LIN {X 0,Y 530.48,Z 461.696,A -85,B 0,C 180,E1 -4342.594,E2 -4342.594} C_VEL
LIN {X 0,Y 530.522,Z 458.64,A -85,B 0,C 180,E1 -4345.082,E2 -4345.082} C_VEL
LIN {X 0,Y 530.512,Z 455.242,A -85,B 0,C 180,E1 -4347.624,E2 -4347.624} C_VEL
LIN {X 0,Y 530.476,Z 451.107,A -85,B 0,C 180,E1 -4350.553,E2 -4350.553} C_VEL
LIN {X 0,Y 530.495,Z 450.409,A -85,B 0,C 180,E1 -4351.109,E2 -4351.109} C_VEL
LIN {X 0,Y 530.816,Z 450.368,A -85,B 0,C 180,E1 -4353.785,E2 -4353.785} C_VEL
LIN {X 0,Y 530.957,Z 450.348,A -85,B 0,C 180,E1 -4356.558,E2 -4356.558} C_VEL
LIN {X 0,Y 530.988,Z 450.346,A -85,B 0,C 180,E1 -4359.443,E2 -4359.443} C_VEL
LIN {X 0,Y 530.985,Z 450.345,A -85,B 0,C 180,E1 -4362.456,E2 -4362.456} C_VEL
LIN {X 0,Y 530.991,Z 450.345,A -85,B 0,C 180,E1 -4365.621,E2 -4365.621} C_VEL
LIN {X 0,Y 530.999,Z 450.345,A -85,B 0,C 180,E1 -4368.565,E2 -4368.565} C_VEL
LIN {X 0,Y 530.986,Z 450.347,A -85,B 0,C 180,E1 -4371.653,E2 -4371.653} C_VEL
LIN {X 0,Y 531.348,Z 452.371,A -85,B 0,C 180,E1 -4372.524,E2 -4372.524} C_VEL
LIN {X 0,Y 532.063,Z 457.513,A -85,B 0,C 180,E1 -4374.465,E2 -4374.465} C_VEL
LIN {X 0,Y 531.885,Z 464.036,A -85,B 0,C 180,E1 -4376.765,E2 -4376.765} C_VEL
LIN {X 0,Y 531.715,Z 471.225,A -85,B 0,C 180,E1 -4379.221,E2 -4379.221} C_VEL
LIN {X 0,Y 531.434,Z 481.002,A -85,B 0,C 180,E1 -4382.428,E2 -4382.428} C_VEL
LIN {X 0,Y 531.236,Z 490.287,A -85,B 0,C 180,E1 -4385.372,E2 -4385.372} C_VEL
LIN {X 0,Y 531.041,Z 500.911,A -85,B 0,C 180,E1 -4388.657,E2 -4388.657} C_VEL
LIN {X 0,Y 530.899,Z 510.447,A -85,B 0,C 180,E1 -4391.475,E2 -4391.475} C_VEL
LIN {X 0,Y 530.798,Z 519.953,A -85,B 0,C 180,E1 -4394.251,E2 -4394.251} C_VEL
LIN {X 0,Y 530.709,Z 527.53,A -85,B 0,C 180,E1 -4396.454,E2 -4396.454} C_VEL
LIN {X 0,Y 532.33,Z 538.348,A -85,B 0,C 180,E1 -4396.739,E2 -4396.739} C_VEL
LIN {X 0,Y 532.122,Z 551.772,A -85,B 0,C 180,E1 -4397.17,E2 -4397.17} C_VEL
LIN {X 0,Y 531.932,Z 563.405,A -85,B 0,C 180,E1 -4397.699,E2 -4397.699} C_VEL
LIN {X 0,Y 531.637,Z 575.806,A -85,B 0,C 180,E1 -4398.441,E2 -4398.441} C_VEL
LIN {X 0,Y 531.384,Z 586.265,A -85,B 0,C 180,E1 -4399.233,E2 -4399.233} C_VEL
LIN {X 0,Y 531.113,Z 595.539,A -85,B 0,C 180,E1 -4400.094,E2 -4400.094} C_VEL
LIN {X 0,Y 530.931,Z 603.991,A -85,B 0,C 180,E1 -4401.052,E2 -4401.052} C_VEL
LIN {X 0,Y 530.758,Z 612.235,A -85,B 0,C 180,E1 -4402.199,E2 -4402.199} C_VEL
LIN {X 0,Y 530.598,Z 619.269,A -85,B 0,C 180,E1 -4403.419,E2 -4403.419} C_VEL
LIN {X 0,Y 530.525,Z 624.949,A -85,B 0,C 180,E1 -4404.679,E2 -4404.679} C_VEL
LIN {X 0,Y 530.522,Z 628.894,A -85,B 0,C 180,E1 -4405.822,E2 -4405.822} C_VEL
LIN {X 0,Y 530.457,Z 631.807,A -85,B 0,C 180,E1 -4406.962,E2 -4406.962} C_VEL
LIN {X 0,Y 530.41,Z 633.194,A -85,B 0,C 180,E1 -4407.722,E2 -4407.722} C_VEL
LIN {X 0,Y 530.344,Z 634.786,A -85,B 0,C 180,E1 -4409.241,E2 -4409.241} C_VEL
LIN {X 0,Y 530.342,Z 635,A -85,B 0,C 180,E1 -4410,E2 -4410} C_VEL
LIN {X 0,Y 530.361,Z 634.184,A -85,B 0,C 180,E1 -4411.519,E2 -4411.519} C_VEL
LIN {X 0,Y 530.41,Z 633.196,A -85,B 0,C 180,E1 -4412.278,E2 -4412.278} C_VEL
LIN {X 0,Y 530.457,Z 631.81,A -85,B 0,C 180,E1 -4413.038,E2 -4413.038} C_VEL
LIN {X 0,Y 530.522,Z 628.895,A -85,B 0,C 180,E1 -4414.178,E2 -4414.178} C_VEL
LIN {X 0,Y 530.525,Z 624.948,A -85,B 0,C 180,E1 -4415.321,E2 -4415.321} C_VEL
LIN {X 0,Y 530.599,Z 619.262,A -85,B 0,C 180,E1 -4416.582,E2 -4416.582} C_VEL
LIN {X 0,Y 530.758,Z 612.235,A -85,B 0,C 180,E1 -4417.801,E2 -4417.801} C_VEL
LIN {X 0,Y 530.931,Z 603.992,A -85,B 0,C 180,E1 -4418.948,E2 -4418.948} C_VEL
LIN {X 0,Y 531.113,Z 595.539,A -85,B 0,C 180,E1 -4419.906,E2 -4419.906} C_VEL
LIN {X 0,Y 531.407,Z 585.091,A -85,B 0,C 180,E1 -4420.863,E2 -4420.863} C_VEL
LIN {X 0,Y 531.675,Z 574.17,A -85,B 0,C 180,E1 -4421.669,E2 -4421.669} C_VEL
LIN {X 0,Y 531.934,Z 563.403,A -85,B 0,C 180,E1 -4422.301,E2 -4422.301} C_VEL
LIN {X 0,Y 532.121,Z 551.762,A -85,B 0,C 180,E1 -4422.83,E2 -4422.83} C_VEL
LIN {X 0,Y 532.301,Z 538.341,A -85,B 0,C 180,E1 -4423.262,E2 -4423.262} C_VEL
LIN {X 0,Y 530.709,Z 527.53,A -85,B 0,C 180,E1 -4423.546,E2 -4423.546} C_VEL
LIN {X 0,Y 530.796,Z 518.456,A -85,B 0,C 180,E1 -4426.144,E2 -4426.144} C_VEL
LIN {X 0,Y 530.89,Z 508.696,A -85,B 0,C 180,E1 -4428.925,E2 -4428.925} C_VEL
LIN {X 0,Y 530.996,Z 498.928,A -85,B 0,C 180,E1 -4431.752,E2 -4431.752} C_VEL
LIN {X 0,Y 531.14,Z 489.323,A -85,B 0,C 180,E1 -4434.633,E2 -4434.633} C_VEL
LIN {X 0,Y 531.316,Z 479.833,A -85,B 0,C 180,E1 -4437.579,E2 -4437.579} C_VEL
LIN {X 0,Y 531.57,Z 470.273,A -85,B 0,C 180,E1 -4440.753,E2 -4440.753} C_VEL
LIN {X 0,Y 531.852,Z 462.239,A -85,B 0,C 180,E1 -4443.711,E2 -4443.711} C_VEL
LIN {X 0,Y 532.105,Z 457.83,A -85,B 0,C 180,E1 -4445.532,E2 -4445.532} C_VEL
LIN {X 0,Y 531.614,Z 453.789,A -85,B 0,C 180,E1 -4447.514,E2 -4447.514} C_VEL
LIN {X 0,Y 531.008,Z 450.344,A -85,B 0,C 180,E1 -4449.647,E2 -4449.647} C_VEL
LIN {X 0,Y 530.981,Z 450.348,A -85,B 0,C 180,E1 -4452.457,E2 -4452.457} C_VEL
LIN {X 0,Y 530.991,Z 450.345,A -85,B 0,C 180,E1 -4455.621,E2 -4455.621} C_VEL
LIN {X 0,Y 531.004,Z 450.345,A -85,B 0,C 180,E1 -4458.565,E2 -4458.565} C_VEL
LIN {X 0,Y 530.963,Z 450.349,A -85,B 0,C 180,E1 -4461.53,E2 -4461.53} C_VEL
LIN {X 0,Y 530.919,Z 450.356,A -85,B 0,C 180,E1 -4464.377,E2 -4464.377} C_VEL
LIN {X 0,Y 530.913,Z 452.045,A -85,B 0,C 180,E1 -4466.509,E2 -4466.509} C_VEL
LIN {X 0,Y 530.832,Z 454.654,A -85,B 0,C 180,E1 -4469.382,E2 -4469.382} C_VEL
LIN {X 0,Y 530.735,Z 457.625,A -85,B 0,C 180,E1 -4472.526,E2 -4472.526} C_VEL
LIN {X 0,Y 530.651,Z 459.965,A -85,B 0,C 180,E1 -4474.925,E2 -4474.925} C_VEL
LIN {X 0,Y 530.573,Z 462.447,A -85,B 0,C 180,E1 -4477.41,E2 -4477.41} C_VEL
LIN {X 0,Y 530.541,Z 465.283,A -85,B 0,C 180,E1 -4480.141,E2 -4480.141} C_VEL
LIN {X 0,Y 530.501,Z 468.236,A -85,B 0,C 180,E1 -4483.055,E2 -4483.055} C_VEL
LIN {X 0,Y 530.487,Z 470.731,A -85,B 0,C 180,E1 -4485.421,E2 -4485.421} C_VEL
LIN {X 0,Y 530.43,Z 471.979,A -85,B 0,C 180,E1 -4486.569,E2 -4486.569} C_VEL
LIN {X 0,Y 532.262,Z 483.592,A -85,B 0,C 180,E1 -4486.931,E2 -4486.931} C_VEL
LIN {X 0,Y 532.044,Z 496.462,A -85,B 0,C 180,E1 -4487.411,E2 -4487.411} C_VEL
LIN {X 0,Y 531.831,Z 508.162,A -85,B 0,C 180,E1 -4488.004,E2 -4488.004} C_VEL
LIN {X 0,Y 531.556,Z 519.593,A -85,B 0,C 180,E1 -4488.754,E2 -4488.754} C_VEL
LIN {X 0,Y 531.258,Z 530.105,A -85,B 0,C 180,E1 -4489.616,E2 -4489.616} C_VEL
LIN {X 0,Y 531.07,Z 538.698,A -85,B 0,C 180,E1 -4490.478,E2 -4490.478} C_VEL
LIN {X 0,Y 530.891,Z 546.614,A -85,B 0,C 180,E1 -4491.435,E2 -4491.435} C_VEL
LIN {X 0,Y 530.69,Z 554.36,A -85,B 0,C 180,E1 -4492.581,E2 -4492.581} C_VEL
LIN {X 0,Y 530.606,Z 561.466,A -85,B 0,C 180,E1 -4493.918,E2 -4493.918} C_VEL
LIN {X 0,Y 530.459,Z 566.204,A -85,B 0,C 180,E1 -4495.06,E2 -4495.06} C_VEL
LIN {X 0,Y 530.516,Z 569.835,A -85,B 0,C 180,E1 -4496.202,E2 -4496.202} C_VEL
LIN {X 0,Y 530.457,Z 571.711,A -85,B 0,C 180,E1 -4496.962,E2 -4496.962} C_VEL
LIN {X 0,Y 530.41,Z 573.13,A -85,B 0,C 180,E1 -4497.722,E2 -4497.722} C_VEL
LIN {X 0,Y 530.344,Z 574.758,A -85,B 0,C 180,E1 -4499.241,E2 -4499.241} C_VEL
LIN {X 0,Y 530.343,Z 574.997,A -85,B 0,C 180,E1 -4500,E2 -4500} C_VEL
LIN {X 0,Y 530.344,Z 574.814,A -85,B 0,C 180,E1 -4500.759,E2 -4500.759} C_VEL
LIN {X 0,Y 530.41,Z 573.26,A -85,B 0,C 180,E1 -4502.278,E2 -4502.278} C_VEL
LIN {X 0,Y 530.458,Z 571.898,A -85,B 0,C 180,E1 -4503.038,E2 -4503.038} C_VEL
LIN {X 0,Y 530.523,Z 569.02,A -85,B 0,C 180,E1 -4504.178,E2 -4504.178} C_VEL
LIN {X 0,Y 530.523,Z 565.117,A -85,B 0,C 180,E1 -4505.321,E2 -4505.321} C_VEL
LIN {X 0,Y 530.605,Z 559.088,A -85,B 0,C 180,E1 -4506.66,E2 -4506.66} C_VEL
LIN {X 0,Y 530.758,Z 552.523,A -85,B 0,C 180,E1 -4507.801,E2 -4507.801} C_VEL
LIN {X 0,Y 530.903,Z 544.338,A -85,B 0,C 180,E1 -4508.949,E2 -4508.949} C_VEL
LIN {X 0,Y 531.107,Z 535.966,A -85,B 0,C 180,E1 -4509.906,E2 -4509.906} C_VEL
LIN {X 0,Y 531.398,Z 525.635,A -85,B 0,C 180,E1 -4510.863,E2 -4510.863} C_VEL
LIN {X 0,Y 531.652,Z 513.899,A -85,B 0,C 180,E1 -4511.732,E2 -4511.732} C_VEL
LIN {X 0,Y 531.904,Z 502.41,A -85,B 0,C 180,E1 -4512.399,E2 -4512.399} C_VEL
LIN {X 0,Y 532.134,Z 490.389,A -85,B 0,C 180,E1 -4512.927,E2 -4512.927} C_VEL
LIN {X 0,Y 532.087,Z 481.415,A -85,B 0,C 180,E1 -4513.231,E2 -4513.231} C_VEL
LIN {X 0,Y 530.419,Z 471.776,A -85,B 0,C 180,E1 -4513.53,E2 -4513.53} C_VEL
LIN {X 0,Y 530.446,Z 468.724,A -85,B 0,C 180,E1 -4516.155,E2 -4516.155} C_VEL
LIN {X 0,Y 530.471,Z 465.114,A -85,B 0,C 180,E1 -4519.343,E2 -4519.343} C_VEL
LIN {X 0,Y 530.496,Z 462.221,A -85,B 0,C 180,E1 -4521.973,E2 -4521.973} C_VEL
LIN {X 0,Y 530.529,Z 458.789,A -85,B 0,C 180,E1 -4525.082,E2 -4525.082} C_VEL
LIN {X 0,Y 530.58,Z 455.925,A -85,B 0,C 180,E1 -4527.62,E2 -4527.62} C_VEL
LIN {X 0,Y 530.613,Z 452.636,A -85,B 0,C 180,E1 -4530.579,E2 -4530.579} C_VEL
LIN {X 0,Y 530.649,Z 450.391,A -85,B 0,C 180,E1 -4532.889,E2 -4532.889} C_VEL
LIN {X 0,Y 530.889,Z 450.359,A -85,B 0,C 180,E1 -4534.838,E2 -4534.838} C_VEL
LIN {X 0,Y 530.969,Z 450.344,A -85,B 0,C 180,E1 -4537.508,E2 -4537.508} C_VEL
LIN {X 0,Y 530.984,Z 450.341,A -85,B 0,C 180,E1 -4539.571,E2 -4539.571} C_VEL
LIN {X 0,Y 530.309,Z 450.43,A -85,B 0,C 180,E1 -4540.204,E2 -4540.204} C_VEL
LIN {X 0,Y 527.449,Z 450.783,A -85,B 0,C 180,E1 -4541.232,E2 -4541.232} C_VEL
LIN {X 0,Y 525.038,Z 451.087,A -85,B 0,C 180,E1 -4542.059,E2 -4542.059} C_VEL
LIN {X 0,Y 524.008,Z 451.211,A -85,B 0,C 180,E1 -4542.698,E2 -4542.698} C_VEL
LIN {X 0,Y 523.926,Z 451.22,A -85,B 0,C 180,E1 -4542.914,E2 -4542.914} C_VEL
LIN {X 0,Y 523.941,Z 451.223,A -85,B 0,C 180,E1 -4545.772,E2 -4545.772} C_VEL
LIN {X 0,Y 523.944,Z 451.223,A -85,B 0,C 180,E1 -4548.908,E2 -4548.908} C_VEL
LIN {X 0,Y 523.92,Z 451.222,A -85,B 0,C 180,E1 -4551.898,E2 -4551.898} C_VEL
LIN {X 0,Y 523.931,Z 451.219,A -85,B 0,C 180,E1 -4554.911,E2 -4554.911} C_VEL
LIN {X 0,Y 523.941,Z 451.224,A -85,B 0,C 180,E1 -4557.68,E2 -4557.68} C_VEL
LIN {X 0,Y 523.96,Z 451.22,A -85,B 0,C 180,E1 -4560.677,E2 -4560.677} C_VEL
LIN {X 0,Y 523.979,Z 451.214,A -85,B 0,C 180,E1 -4563.729,E2 -4563.729} C_VEL
LIN {X 0,Y 523.918,Z 451.226,A -85,B 0,C 180,E1 -4566.27,E2 -4566.27} C_VEL
LIN {X 0,Y 523.951,Z 451.217,A -85,B 0,C 180,E1 -4568.767,E2 -4568.767} C_VEL
LIN {X 0,Y 523.954,Z 451.221,A -85,B 0,C 180,E1 -4571.221,E2 -4571.221} C_VEL
LIN {X 0,Y 523.936,Z 451.22,A -85,B 0,C 180,E1 -4573.639,E2 -4573.639} C_VEL
LIN {X 0,Y 523.945,Z 451.22,A -85,B 0,C 180,E1 -4576.028,E2 -4576.028} C_VEL
LIN {X 0,Y 524.019,Z 451.211,A -85,B 0,C 180,E1 -4578.394,E2 -4578.394} C_VEL
LIN {X 0,Y 524.007,Z 451.215,A -85,B 0,C 180,E1 -4581.516,E2 -4581.516} C_VEL
LIN {X 0,Y 524.085,Z 451.203,A -85,B 0,C 180,E1 -4584.614,E2 -4584.614} C_VEL
LIN {X 0,Y 524.117,Z 451.197,A -85,B 0,C 180,E1 -4587.694,E2 -4587.694} C_VEL
LIN {X 0,Y 524.128,Z 451.195,A -85,B 0,C 180,E1 -4590.768,E2 -4590.768} C_VEL
LIN {X 0,Y 524.075,Z 451.202,A -85,B 0,C 180,E1 -4593.075,E2 -4593.075} C_VEL
LIN {X 0,Y 524.032,Z 451.208,A -85,B 0,C 180,E1 -4596.159,E2 -4596.159} C_VEL
LIN {X 0,Y 523.993,Z 451.214,A -85,B 0,C 180,E1 -4599.262,E2 -4599.262} C_VEL
LIN {X 0,Y 524.009,Z 451.211,A -85,B 0,C 180,E1 -4601.739,E2 -4601.739} C_VEL
LIN {X 0,Y 524,Z 451.211,A -85,B 0,C 180,E1 -4605.052,E2 -4605.052} C_VEL
LIN {X 0,Y 523.97,Z 451.216,A -85,B 0,C 180,E1 -4607.969,E2 -4607.969} C_VEL
LIN {X 0,Y 523.978,Z 451.217,A -85,B 0,C 180,E1 -4610.41,E2 -4610.41} C_VEL
LIN {X 0,Y 523.916,Z 451.224,A -85,B 0,C 180,E1 -4612.893,E2 -4612.893} C_VEL
LIN {X 0,Y 523.989,Z 451.217,A -85,B 0,C 180,E1 -4616.019,E2 -4616.019} C_VEL
LIN {X 0,Y 523.944,Z 451.219,A -85,B 0,C 180,E1 -4618.875,E2 -4618.875} C_VEL
LIN {X 0,Y 523.927,Z 451.222,A -85,B 0,C 180,E1 -4621.544,E2 -4621.544} C_VEL
LIN {X 0,Y 523.946,Z 451.222,A -85,B 0,C 180,E1 -4624.289,E2 -4624.289} C_VEL
LIN {X 0,Y 523.915,Z 451.221,A -85,B 0,C 180,E1 -4627.132,E2 -4627.132} C_VEL
LIN {X 0,Y 523.942,Z 451.219,A -85,B 0,C 180,E1 -4630.13,E2 -4630.13} C_VEL
LIN {X 0,Y 523.94,Z 451.219,A -85,B 0,C 180,E1 -4632.459,E2 -4632.459} C_VEL
LIN {X 0,Y 523.96,Z 451.218,A -85,B 0,C 180,E1 -4635.309,E2 -4635.309} C_VEL
LIN {X 0,Y 523.964,Z 451.217,A -85,B 0,C 180,E1 -4638.689,E2 -4638.689} C_VEL
LIN {X 0,Y 523.921,Z 451.221,A -85,B 0,C 180,E1 -4641.08,E2 -4641.08} C_VEL
LIN {X 0,Y 523.902,Z 451.225,A -85,B 0,C 180,E1 -4643.825,E2 -4643.825} C_VEL
LIN {X 0,Y 523.735,Z 451.249,A -85,B 0,C 180,E1 -4646.62,E2 -4646.62} C_VEL
LIN {X 0,Y 523.511,Z 451.278,A -85,B 0,C 180,E1 -4648.428,E2 -4648.428} C_VEL
LIN {X 0,Y 523.448,Z 454.349,A -85,B 0,C 180,E1 -4651.095,E2 -4651.095} C_VEL
LIN {X 0,Y 523.469,Z 457.412,A -85,B 0,C 180,E1 -4653.701,E2 -4653.701} C_VEL
LIN {X 0,Y 523.43,Z 460.399,A -85,B 0,C 180,E1 -4656.246,E2 -4656.246} C_VEL
LIN {X 0,Y 523.379,Z 463.33,A -85,B 0,C 180,E1 -4658.742,E2 -4658.742} C_VEL
LIN {X 0,Y 523.377,Z 466.222,A -85,B 0,C 180,E1 -4661.199,E2 -4661.199} C_VEL
LIN {X 0,Y 523.346,Z 468.929,A -85,B 0,C 180,E1 -4663.62,E2 -4663.62} C_VEL
LIN {X 0,Y 523.357,Z 472.059,A -85,B 0,C 180,E1 -4666.383,E2 -4666.383} C_VEL
LIN {X 0,Y 525.327,Z 483.715,A -85,B 0,C 180,E1 -4666.755,E2 -4666.755} C_VEL
LIN {X 0,Y 525.094,Z 496.507,A -85,B 0,C 180,E1 -4667.241,E2 -4667.241} C_VEL
LIN {X 0,Y 524.861,Z 507.803,A -85,B 0,C 180,E1 -4667.82,E2 -4667.82} C_VEL
LIN {X 0,Y 524.658,Z 516.989,A -85,B 0,C 180,E1 -4668.408,E2 -4668.408} C_VEL
LIN {X 0,Y 524.401,Z 525.79,A -85,B 0,C 180,E1 -4669.088,E2 -4669.088} C_VEL
LIN {X 0,Y 524.206,Z 533.214,A -85,B 0,C 180,E1 -4669.767,E2 -4669.767} C_VEL
LIN {X 0,Y 524.011,Z 540.446,A -85,B 0,C 180,E1 -4670.543,E2 -4670.543} C_VEL
LIN {X 0,Y 523.825,Z 548.025,A -85,B 0,C 180,E1 -4671.513,E2 -4671.513} C_VEL
LIN {X 0,Y 523.637,Z 554.324,A -85,B 0,C 180,E1 -4672.48,E2 -4672.48} C_VEL
LIN {X 0,Y 523.527,Z 559.403,A -85,B 0,C 180,E1 -4673.416,E2 -4673.416} C_VEL
LIN {X 0,Y 523.521,Z 563.128,A -85,B 0,C 180,E1 -4674.221,E2 -4674.221} C_VEL
LIN {X 0,Y 523.366,Z 567.47,A -85,B 0,C 180,E1 -4675.378,E2 -4675.378} C_VEL
LIN {X 0,Y 523.444,Z 569.845,A -85,B 0,C 180,E1 -4676.15,E2 -4676.15} C_VEL
LIN {X 0,Y 523.368,Z 571.665,A -85,B 0,C 180,E1 -4676.921,E2 -4676.921} C_VEL
LIN {X 0,Y 523.274,Z 574.132,A -85,B 0,C 180,E1 -4678.461,E2 -4678.461} C_VEL
LIN {X 0,Y 523.251,Z 574.741,A -85,B 0,C 180,E1 -4679.23,E2 -4679.23} C_VEL
LIN {X 0,Y 523.25,Z 574.79,A -85,B 0,C 180,E1 -4680.769,E2 -4680.769} C_VEL
LIN {X 0,Y 523.275,Z 574.222,A -85,B 0,C 180,E1 -4681.539,E2 -4681.539} C_VEL
LIN {X 0,Y 523.368,Z 571.857,A -85,B 0,C 180,E1 -4683.079,E2 -4683.079} C_VEL
LIN {X 0,Y 523.441,Z 568.971,A -85,B 0,C 180,E1 -4684.235,E2 -4684.235} C_VEL
LIN {X 0,Y 523.463,Z 565.052,A -85,B 0,C 180,E1 -4685.393,E2 -4685.393} C_VEL
LIN {X 0,Y 523.468,Z 561.285,A -85,B 0,C 180,E1 -4686.291,E2 -4686.291} C_VEL
LIN {X 0,Y 523.595,Z 556.013,A -85,B 0,C 180,E1 -4687.326,E2 -4687.326} C_VEL
LIN {X 0,Y 523.756,Z 550.051,A -85,B 0,C 180,E1 -4688.294,E2 -4688.294} C_VEL
LIN {X 0,Y 523.901,Z 542.867,A -85,B 0,C 180,E1 -4689.263,E2 -4689.263} C_VEL
LIN {X 0,Y 524.105,Z 536.073,A -85,B 0,C 180,E1 -4690.039,E2 -4690.039} C_VEL
LIN {X 0,Y 524.367,Z 526.894,A -85,B 0,C 180,E1 -4690.913,E2 -4690.913} C_VEL
LIN {X 0,Y 524.647,Z 516.967,A -85,B 0,C 180,E1 -4691.688,E2 -4691.688} C_VEL
LIN {X 0,Y 524.902,Z 506.164,A -85,B 0,C 180,E1 -4692.37,E2 -4692.37} C_VEL
LIN {X 0,Y 525.174,Z 492.987,A -85,B 0,C 180,E1 -4693.002,E2 -4693.002} C_VEL
LIN {X 0,Y 525.167,Z 482.311,A -85,B 0,C 180,E1 -4693.381,E2 -4693.381} C_VEL
LIN {X 0,Y 523.368,Z 472.349,A -85,B 0,C 180,E1 -4693.69,E2 -4693.69} C_VEL
LIN {X 0,Y 523.394,Z 469.456,A -85,B 0,C 180,E1 -4696.378,E2 -4696.378} C_VEL
LIN {X 0,Y 523.404,Z 466.652,A -85,B 0,C 180,E1 -4698.8,E2 -4698.8} C_VEL
LIN {X 0,Y 523.389,Z 463.847,A -85,B 0,C 180,E1 -4701.257,E2 -4701.257} C_VEL
LIN {X 0,Y 523.446,Z 460.496,A -85,B 0,C 180,E1 -4704.077,E2 -4704.077} C_VEL
LIN {X 0,Y 523.464,Z 457.622,A -85,B 0,C 180,E1 -4706.299,E2 -4706.299} C_VEL
LIN {X 0,Y 523.424,Z 453.629,A -85,B 0,C 180,E1 -4709.219,E2 -4709.219} C_VEL
LIN {X 0,Y 523.415,Z 451.397,A -85,B 0,C 180,E1 -4710.757,E2 -4710.757} C_VEL
LIN {X 0,Y 523.775,Z 451.245,A -85,B 0,C 180,E1 -4713.704,E2 -4713.704} C_VEL
LIN {X 0,Y 523.905,Z 451.226,A -85,B 0,C 180,E1 -4716.401,E2 -4716.401} C_VEL
LIN {X 0,Y 523.922,Z 451.224,A -85,B 0,C 180,E1 -4719.085,E2 -4719.085} C_VEL
LIN {X 0,Y 523.959,Z 451.222,A -85,B 0,C 180,E1 -4722.118,E2 -4722.118} C_VEL
LIN {X 0,Y 523.959,Z 451.219,A -85,B 0,C 180,E1 -4725.309,E2 -4725.309} C_VEL
LIN {X 0,Y 523.961,Z 451.221,A -85,B 0,C 180,E1 -4728.689,E2 -4728.689} C_VEL
LIN {X 0,Y 523.949,Z 451.354,A -85,B 0,C 180,E1 -4731.534,E2 -4731.534} C_VEL
LIN {X 0,Y 525.005,Z 457.462,A -85,B 0,C 180,E1 -4733.913,E2 -4733.913} C_VEL
LIN {X 0,Y 525.021,Z 463.46,A -85,B 0,C 180,E1 -4736.093,E2 -4736.093} C_VEL
LIN {X 0,Y 524.745,Z 471.821,A -85,B 0,C 180,E1 -4739,E2 -4739} C_VEL
LIN {X 0,Y 524.455,Z 481.344,A -85,B 0,C 180,E1 -4742.183,E2 -4742.183} C_VEL
LIN {X 0,Y 524.195,Z 491.457,A -85,B 0,C 180,E1 -4745.441,E2 -4745.441} C_VEL
LIN {X 0,Y 523.995,Z 500.755,A -85,B 0,C 180,E1 -4748.356,E2 -4748.356} C_VEL
LIN {X 0,Y 523.837,Z 510.21,A -85,B 0,C 180,E1 -4751.216,E2 -4751.216} C_VEL
LIN {X 0,Y 523.722,Z 519.719,A -85,B 0,C 180,E1 -4754.032,E2 -4754.032} C_VEL
LIN {X 0,Y 523.658,Z 527.602,A -85,B 0,C 180,E1 -4756.293,E2 -4756.293} C_VEL
LIN {X 0,Y 525.397,Z 538.948,A -85,B 0,C 180,E1 -4756.585,E2 -4756.585} C_VEL
LIN {X 0,Y 525.195,Z 551.519,A -85,B 0,C 180,E1 -4756.998,E2 -4756.998} C_VEL
LIN {X 0,Y 524.981,Z 563.233,A -85,B 0,C 180,E1 -4757.534,E2 -4757.534} C_VEL
LIN {X 0,Y 524.696,Z 574.33,A -85,B 0,C 180,E1 -4758.191,E2 -4758.191} C_VEL
LIN {X 0,Y 524.431,Z 585.079,A -85,B 0,C 180,E1 -4758.991,E2 -4758.991} C_VEL
LIN {X 0,Y 524.094,Z 595.539,A -85,B 0,C 180,E1 -4759.96,E2 -4759.96} C_VEL
LIN {X 0,Y 523.896,Z 603.992,A -85,B 0,C 180,E1 -4760.931,E2 -4760.931} C_VEL
LIN {X 0,Y 523.688,Z 612.234,A -85,B 0,C 180,E1 -4762.093,E2 -4762.093} C_VEL
LIN {X 0,Y 523.574,Z 617.868,A -85,B 0,C 180,E1 -4763.061,E2 -4763.061} C_VEL
LIN {X 0,Y 523.544,Z 623.366,A -85,B 0,C 180,E1 -4764.222,E2 -4764.222} C_VEL
LIN {X 0,Y 523.361,Z 627.677,A -85,B 0,C 180,E1 -4765.379,E2 -4765.379} C_VEL
LIN {X 0,Y 523.443,Z 629.958,A -85,B 0,C 180,E1 -4766.151,E2 -4766.151} C_VEL
LIN {X 0,Y 523.367,Z 631.807,A -85,B 0,C 180,E1 -4766.921,E2 -4766.921} C_VEL
LIN {X 0,Y 523.334,Z 633.193,A -85,B 0,C 180,E1 -4767.691,E2 -4767.691} C_VEL
LIN {X 0,Y 523.25,Z 634.785,A -85,B 0,C 180,E1 -4769.23,E2 -4769.23} C_VEL
LIN {X 0,Y 523.246,Z 635,A -85,B 0,C 180,E1 -4770,E2 -4770} C_VEL
LIN {X 0,Y 523.274,Z 634.183,A -85,B 0,C 180,E1 -4771.539,E2 -4771.539} C_VEL
LIN {X 0,Y 523.334,Z 633.196,A -85,B 0,C 180,E1 -4772.309,E2 -4772.309} C_VEL
LIN {X 0,Y 523.367,Z 631.81,A -85,B 0,C 180,E1 -4773.079,E2 -4773.079} C_VEL
LIN {X 0,Y 523.441,Z 628.895,A -85,B 0,C 180,E1 -4774.235,E2 -4774.235} C_VEL
LIN {X 0,Y 523.464,Z 624.948,A -85,B 0,C 180,E1 -4775.393,E2 -4775.393} C_VEL
LIN {X 0,Y 523.523,Z 619.726,A -85,B 0,C 180,E1 -4776.581,E2 -4776.581} C_VEL
LIN {X 0,Y 523.665,Z 613.466,A -85,B 0,C 180,E1 -4777.713,E2 -4777.713} C_VEL
LIN {X 0,Y 523.857,Z 605.477,A -85,B 0,C 180,E1 -4778.875,E2 -4778.875} C_VEL
LIN {X 0,Y 524.085,Z 597.332,A -85,B 0,C 180,E1 -4779.845,E2 -4779.845} C_VEL
LIN {X 0,Y 524.363,Z 587.393,A -85,B 0,C 180,E1 -4780.815,E2 -4780.815} C_VEL
LIN {X 0,Y 524.611,Z 577.516,A -85,B 0,C 180,E1 -4781.593,E2 -4781.593} C_VEL
LIN {X 0,Y 524.886,Z 566.02,A -85,B 0,C 180,E1 -4782.312,E2 -4782.312} C_VEL
LIN {X 0,Y 525.102,Z 553.772,A -85,B 0,C 180,E1 -4782.906,E2 -4782.906} C_VEL
LIN {X 0,Y 525.36,Z 540.627,A -85,B 0,C 180,E1 -4783.367,E2 -4783.367} C_VEL
LIN {X 0,Y 524.994,Z 536.001,A -85,B 0,C 180,E1 -4783.499,E2 -4783.499} C_VEL
LIN {X 0,Y 523.642,Z 527.15,A -85,B 0,C 180,E1 -4783.733,E2 -4783.733} C_VEL
LIN {X 0,Y 523.699,Z 517.982,A -85,B 0,C 180,E1 -4786.369,E2 -4786.369} C_VEL
LIN {X 0,Y 523.809,Z 508.216,A -85,B 0,C 180,E1 -4789.191,E2 -4789.191} C_VEL
LIN {X 0,Y 523.928,Z 499.908,A -85,B 0,C 180,E1 -4791.647,E2 -4791.647} C_VEL
LIN {X 0,Y 524.071,Z 490.306,A -85,B 0,C 180,E1 -4794.565,E2 -4794.565} C_VEL
LIN {X 0,Y 524.266,Z 481.195,A -85,B 0,C 180,E1 -4797.446,E2 -4797.446} C_VEL
LIN {X 0,Y 524.536,Z 471.859,A -85,B 0,C 180,E1 -4800.607,E2 -4800.607} C_VEL
LIN {X 0,Y 524.813,Z 464.622,A -85,B 0,C 180,E1 -4803.302,E2 -4803.302} C_VEL
LIN {X 0,Y 525.135,Z 459.841,A -85,B 0,C 180,E1 -4805.276,E2 -4805.276} C_VEL
LIN {X 0,Y 524.825,Z 456.188,A -85,B 0,C 180,E1 -4807.057,E2 -4807.057} C_VEL
LIN {X 0,Y 524.241,Z 452.777,A -85,B 0,C 180,E1 -4809.057,E2 -4809.057} C_VEL
LIN {X 0,Y 523.956,Z 451.222,A -85,B 0,C 180,E1 -4810.33,E2 -4810.33} C_VEL
LIN {X 0,Y 523.924,Z 451.226,A -85,B 0,C 180,E1 -4813.167,E2 -4813.167} C_VEL
LIN {X 0,Y 523.945,Z 451.223,A -85,B 0,C 180,E1 -4815.772,E2 -4815.772} C_VEL
LIN {X 0,Y 523.948,Z 451.223,A -85,B 0,C 180,E1 -4818.908,E2 -4818.908} C_VEL
LIN {X 0,Y 523.92,Z 451.227,A -85,B 0,C 180,E1 -4821.898,E2 -4821.898} C_VEL
LIN {X 0,Y 523.874,Z 451.233,A -85,B 0,C 180,E1 -4823.823,E2 -4823.823} C_VEL
LIN {X 0,Y 523.901,Z 451.733,A -85,B 0,C 180,E1 -4824.915,E2 -4824.915} C_VEL
LIN {X 0,Y 523.851,Z 454.069,A -85,B 0,C 180,E1 -4827.695,E2 -4827.695} C_VEL
LIN {X 0,Y 523.751,Z 456.345,A -85,B 0,C 180,E1 -4830.232,E2 -4830.232} C_VEL
LIN {X 0,Y 523.659,Z 458.772,A -85,B 0,C 180,E1 -4832.851,E2 -4832.851} C_VEL
LIN {X 0,Y 523.603,Z 461.709,A -85,B 0,C 180,E1 -4835.885,E2 -4835.885} C_VEL
LIN {X 0,Y 523.502,Z 464.558,A -85,B 0,C 180,E1 -4838.748,E2 -4838.748} C_VEL
LIN {X 0,Y 523.444,Z 467.092,A -85,B 0,C 180,E1 -4841.202,E2 -4841.202} C_VEL
LIN {X 0,Y 523.42,Z 469.54,A -85,B 0,C 180,E1 -4843.622,E2 -4843.622} C_VEL
LIN {X 0,Y 523.39,Z 472.501,A -85,B 0,C 180,E1 -4846.409,E2 -4846.409} C_VEL
LIN {X 0,Y 525.351,Z 483.781,A -85,B 0,C 180,E1 -4846.756,E2 -4846.756} C_VEL
LIN {X 0,Y 525.115,Z 496.677,A -85,B 0,C 180,E1 -4847.242,E2 -4847.242} C_VEL
LIN {X 0,Y 524.907,Z 507.589,A -85,B 0,C 180,E1 -4847.797,E2 -4847.797} C_VEL
LIN {X 0,Y 524.617,Z 518.543,A -85,B 0,C 180,E1 -4848.506,E2 -4848.506} C_VEL
LIN {X 0,Y 524.298,Z 529.248,A -85,B 0,C 180,E1 -4849.379,E2 -4849.379} C_VEL
LIN {X 0,Y 524.059,Z 538.866,A -85,B 0,C 180,E1 -4850.35,E2 -4850.35} C_VEL
LIN {X 0,Y 523.859,Z 546.736,A -85,B 0,C 180,E1 -4851.319,E2 -4851.319} C_VEL
LIN {X 0,Y 523.637,Z 554.426,A -85,B 0,C 180,E1 -4852.481,E2 -4852.481} C_VEL
LIN {X 0,Y 523.519,Z 561.469,A -85,B 0,C 180,E1 -4853.835,E2 -4853.835} C_VEL
LIN {X 0,Y 523.384,Z 566.206,A -85,B 0,C 180,E1 -4854.993,E2 -4854.993} C_VEL
LIN {X 0,Y 523.444,Z 569.836,A -85,B 0,C 180,E1 -4856.151,E2 -4856.151} C_VEL
LIN {X 0,Y 523.368,Z 571.713,A -85,B 0,C 180,E1 -4856.921,E2 -4856.921} C_VEL
LIN {X 0,Y 523.334,Z 573.13,A -85,B 0,C 180,E1 -4857.691,E2 -4857.691} C_VEL
LIN {X 0,Y 523.25,Z 574.758,A -85,B 0,C 180,E1 -4859.231,E2 -4859.231} C_VEL
LIN {X 0,Y 523.247,Z 574.997,A -85,B 0,C 180,E1 -4860,E2 -4860} C_VEL
LIN {X 0,Y 523.25,Z 574.813,A -85,B 0,C 180,E1 -4860.77,E2 -4860.77} C_VEL
LIN {X 0,Y 523.334,Z 573.258,A -85,B 0,C 180,E1 -4862.309,E2 -4862.309} C_VEL
LIN {X 0,Y 523.368,Z 571.896,A -85,B 0,C 180,E1 -4863.079,E2 -4863.079} C_VEL
LIN {X 0,Y 523.441,Z 569.018,A -85,B 0,C 180,E1 -4864.235,E2 -4864.235} C_VEL
LIN {X 0,Y 523.462,Z 565.115,A -85,B 0,C 180,E1 -4865.393,E2 -4865.393} C_VEL
LIN {X 0,Y 523.529,Z 559.48,A -85,B 0,C 180,E1 -4866.673,E2 -4866.673} C_VEL
LIN {X 0,Y 523.691,Z 552.578,A -85,B 0,C 180,E1 -4867.907,E2 -4867.907} C_VEL
LIN {X 0,Y 523.868,Z 544.443,A -85,B 0,C 180,E1 -4869.07,E2 -4869.07} C_VEL
LIN {X 0,Y 524.097,Z 536.101,A -85,B 0,C 180,E1 -4870.04,E2 -4870.04} C_VEL
LIN {X 0,Y 524.42,Z 525.787,A -85,B 0,C 180,E1 -4871.01,E2 -4871.01} C_VEL
LIN {X 0,Y 524.68,Z 514.638,A -85,B 0,C 180,E1 -4871.851,E2 -4871.851} C_VEL
LIN {X 0,Y 524.925,Z 504.379,A -85,B 0,C 180,E1 -4872.468,E2 -4872.468} C_VEL
LIN {X 0,Y 525.17,Z 493.04,A -85,B 0,C 180,E1 -4873.003,E2 -4873.003} C_VEL
LIN {X 0,Y 525.171,Z 482.319,A -85,B 0,C 180,E1 -4873.384,E2 -4873.384} C_VEL
LIN {X 0,Y 523.366,Z 472.121,A -85,B 0,C 180,E1 -4873.691,E2 -4873.691} C_VEL
LIN {X 0,Y 523.359,Z 469.005,A -85,B 0,C 180,E1 -4876.38,E2 -4876.38} C_VEL
LIN {X 0,Y 523.406,Z 465.387,A -85,B 0,C 180,E1 -4879.615,E2 -4879.615} C_VEL
LIN {X 0,Y 523.438,Z 462.669,A -85,B 0,C 180,E1 -4882.113,E2 -4882.113} C_VEL
LIN {X 0,Y 523.433,Z 459.915,A -85,B 0,C 180,E1 -4884.597,E2 -4884.597} C_VEL
LIN {X 0,Y 523.514,Z 457.055,A -85,B 0,C 180,E1 -4887.158,E2 -4887.158} C_VEL
LIN {X 0,Y 523.522,Z 454.153,A -85,B 0,C 180,E1 -4889.783,E2 -4889.783} C_VEL
LIN {X 0,Y 523.556,Z 451.273,A -85,B 0,C 180,E1 -4892.476,E2 -4892.476} C_VEL
LIN {X 0,Y 523.857,Z 451.233,A -85,B 0,C 180,E1 -4895.232,E2 -4895.232} C_VEL
LIN {X 0,Y 523.92,Z 451.222,A -85,B 0,C 180,E1 -4898.102,E2 -4898.102} C_VEL
LIN {X 0,Y 523.946,Z 451.217,A -85,B 0,C 180,E1 -4901.092,E2 -4901.092} C_VEL
LIN {X 0,Y 523.926,Z 451.22,A -85,B 0,C 180,E1 -4902.914,E2 -4902.914} C_VEL
LIN {X 0,Y 523.268,Z 451.306,A -85,B 0,C 180,E1 -4903.556,E2 -4903.556} C_VEL
LIN {X 0,Y 520.427,Z 451.658,A -85,B 0,C 180,E1 -4904.598,E2 -4904.598} C_VEL
LIN {X 0,Y 518.013,Z 451.961,A -85,B 0,C 180,E1 -4905.438,E2 -4905.438} C_VEL
LIN {X 0,Y 516.965,Z 452.089,A -85,B 0,C 180,E1 -4906.086,E2 -4906.086} C_VEL
LIN {X 0,Y 516.873,Z 452.099,A -85,B 0,C 180,E1 -4906.305,E2 -4906.305} C_VEL
LIN {X 0,Y 516.888,Z 452.101,A -85,B 0,C 180,E1 -4909.258,E2 -4909.258} C_VEL
LIN {X 0,Y 516.868,Z 452.104,A -85,B 0,C 180,E1 -4912.274,E2 -4912.274} C_VEL
LIN {X 0,Y 516.89,Z 452.097,A -85,B 0,C 180,E1 -4915.176,E2 -4915.176} C_VEL
LIN {X 0,Y 516.879,Z 452.101,A -85,B 0,C 180,E1 -4917.975,E2 -4917.975} C_VEL
LIN {X 0,Y 516.927,Z 452.096,A -85,B 0,C 180,E1 -4920.696,E2 -4920.696} C_VEL
LIN {X 0,Y 516.948,Z 452.09,A -85,B 0,C 180,E1 -4923.804,E2 -4923.804} C_VEL
LIN {X 0,Y 516.865,Z 452.1,A -85,B 0,C 180,E1 -4926.776,E2 -4926.776} C_VEL
LIN {X 0,Y 516.945,Z 452.095,A -85,B 0,C 180,E1 -4929.732,E2 -4929.732} C_VEL
LIN {X 0,Y 516.913,Z 452.097,A -85,B 0,C 180,E1 -4932.596,E2 -4932.596} C_VEL
LIN {X 0,Y 516.949,Z 452.093,A -85,B 0,C 180,E1 -4935.03,E2 -4935.03} C_VEL
LIN {X 0,Y 516.972,Z 452.091,A -85,B 0,C 180,E1 -4938.234,E2 -4938.234} C_VEL
LIN {X 0,Y 516.971,Z 452.09,A -85,B 0,C 180,E1 -4941.4,E2 -4941.4} C_VEL
LIN {X 0,Y 517.016,Z 452.083,A -85,B 0,C 180,E1 -4943.757,E2 -4943.757} C_VEL
LIN {X 0,Y 517.09,Z 452.072,A -85,B 0,C 180,E1 -4947.663,E2 -4947.663} C_VEL
LIN {X 0,Y 517.098,Z 452.07,A -85,B 0,C 180,E1 -4950.779,E2 -4950.779} C_VEL
LIN {X 0,Y 517.016,Z 452.082,A -85,B 0,C 180,E1 -4953.117,E2 -4953.117} C_VEL
LIN {X 0,Y 516.995,Z 452.084,A -85,B 0,C 180,E1 -4956.243,E2 -4956.243} C_VEL
LIN {X 0,Y 516.949,Z 452.09,A -85,B 0,C 180,E1 -4959.389,E2 -4959.389} C_VEL
LIN {X 0,Y 516.959,Z 452.09,A -85,B 0,C 180,E1 -4961.807,E2 -4961.807} C_VEL
LIN {X 0,Y 516.951,Z 452.09,A -85,B 0,C 180,E1 -4965.146,E2 -4965.146} C_VEL
LIN {X 0,Y 516.931,Z 452.092,A -85,B 0,C 180,E1 -4968.222,E2 -4968.222} C_VEL
LIN {X 0,Y 516.918,Z 452.098,A -85,B 0,C 180,E1 -4970.701,E2 -4970.701} C_VEL
LIN {X 0,Y 516.897,Z 452.101,A -85,B 0,C 180,E1 -4974.073,E2 -4974.073} C_VEL
LIN {X 0,Y 516.928,Z 452.091,A -85,B 0,C 180,E1 -4976.658,E2 -4976.658} C_VEL
LIN {X 0,Y 516.917,Z 452.099,A -85,B 0,C 180,E1 -4979.524,E2 -4979.524} C_VEL
LIN {X 0,Y 516.901,Z 452.1,A -85,B 0,C 180,E1 -4982.543,E2 -4982.543} C_VEL
LIN {X 0,Y 516.884,Z 452.098,A -85,B 0,C 180,E1 -4985.332,E2 -4985.332} C_VEL
LIN {X 0,Y 516.885,Z 452.103,A -85,B 0,C 180,E1 -4987.943,E2 -4987.943} C_VEL
LIN {X 0,Y 516.888,Z 452.097,A -85,B 0,C 180,E1 -4990.742,E2 -4990.742} C_VEL
LIN {X 0,Y 516.887,Z 452.101,A -85,B 0,C 180,E1 -4992.831,E2 -4992.831} C_VEL
LIN {X 0,Y 516.928,Z 452.097,A -85,B 0,C 180,E1 -4995.01,E2 -4995.01} C_VEL
LIN {X 0,Y 516.921,Z 452.097,A -85,B 0,C 180,E1 -4998.398,E2 -4998.398} C_VEL
LIN {X 0,Y 516.884,Z 452.099,A -85,B 0,C 180,E1 -5001.284,E2 -5001.284} C_VEL
LIN {X 0,Y 516.829,Z 452.104,A -85,B 0,C 180,E1 -5004.216,E2 -5004.216} C_VEL
LIN {X 0,Y 516.649,Z 452.132,A -85,B 0,C 180,E1 -5007.035,E2 -5007.035} C_VEL
LIN {X 0,Y 516.413,Z 452.46,A -85,B 0,C 180,E1 -5009.024,E2 -5009.024} C_VEL
LIN {X 0,Y 516.413,Z 456.225,A -85,B 0,C 180,E1 -5012.203,E2 -5012.203} C_VEL
LIN {X 0,Y 516.395,Z 458.54,A -85,B 0,C 180,E1 -5014.182,E2 -5014.182} C_VEL
LIN {X 0,Y 516.337,Z 461.541,A -85,B 0,C 180,E1 -5016.751,E2 -5016.751} C_VEL
LIN {X 0,Y 516.359,Z 465.42,A -85,B 0,C 180,E1 -5020.107,E2 -5020.107} C_VEL
LIN {X 0,Y 516.315,Z 468.277,A -85,B 0,C 180,E1 -5022.574,E2 -5022.574} C_VEL
LIN {X 0,Y 516.284,Z 471.96,A -85,B 0,C 180,E1 -5025.816,E2 -5025.816} C_VEL
LIN {X 0,Y 516.315,Z 472.429,A -85,B 0,C 180,E1 -5026.219,E2 -5026.219} C_VEL
LIN {X 0,Y 518.431,Z 484.572,A -85,B 0,C 180,E1 -5026.601,E2 -5026.601} C_VEL
LIN {X 0,Y 518.147,Z 497.723,A -85,B 0,C 180,E1 -5027.117,E2 -5027.117} C_VEL
LIN {X 0,Y 517.916,Z 508.695,A -85,B 0,C 180,E1 -5027.695,E2 -5027.695} C_VEL
LIN {X 0,Y 517.635,Z 519.958,A -85,B 0,C 180,E1 -5028.447,E2 -5028.447} C_VEL
LIN {X 0,Y 517.26,Z 531.51,A -85,B 0,C 180,E1 -5029.43,E2 -5029.43} C_VEL
LIN {X 0,Y 517.006,Z 540.749,A -85,B 0,C 180,E1 -5030.414,E2 -5030.414} C_VEL
LIN {X 0,Y 516.806,Z 548.349,A -85,B 0,C 180,E1 -5031.397,E2 -5031.397} C_VEL
LIN {X 0,Y 516.563,Z 555.827,A -85,B 0,C 180,E1 -5032.573,E2 -5032.573} C_VEL
LIN {X 0,Y 516.453,Z 561.8,A -85,B 0,C 180,E1 -5033.75,E2 -5033.75} C_VEL
LIN {X 0,Y 516.318,Z 566.515,A -85,B 0,C 180,E1 -5034.924,E2 -5034.924} C_VEL
LIN {X 0,Y 516.373,Z 570.116,A -85,B 0,C 180,E1 -5036.098,E2 -5036.098} C_VEL
LIN {X 0,Y 516.283,Z 571.936,A -85,B 0,C 180,E1 -5036.878,E2 -5036.878} C_VEL
LIN {X 0,Y 516.191,Z 574.389,A -85,B 0,C 180,E1 -5038.439,E2 -5038.439} C_VEL
LIN {X 0,Y 516.161,Z 574.994,A -85,B 0,C 180,E1 -5039.22,E2 -5039.22} C_VEL
LIN {X 0,Y 516.16,Z 575.045,A -85,B 0,C 180,E1 -5040.78,E2 -5040.78} C_VEL
LIN {X 0,Y 516.192,Z 574.489,A -85,B 0,C 180,E1 -5041.56,E2 -5041.56} C_VEL
LIN {X 0,Y 516.283,Z 572.145,A -85,B 0,C 180,E1 -5043.121,E2 -5043.121} C_VEL
LIN {X 0,Y 516.36,Z 569.294,A -85,B 0,C 180,E1 -5044.293,E2 -5044.293} C_VEL
LIN {X 0,Y 516.401,Z 565.421,A -85,B 0,C 180,E1 -5045.467,E2 -5045.467} C_VEL
LIN {X 0,Y 516.477,Z 560.579,A -85,B 0,C 180,E1 -5046.608,E2 -5046.608} C_VEL
LIN {X 0,Y 516.619,Z 554.123,A -85,B 0,C 180,E1 -5047.819,E2 -5047.819} C_VEL
LIN {X 0,Y 516.854,Z 546.266,A -85,B 0,C 180,E1 -5048.996,E2 -5048.996} C_VEL
LIN {X 0,Y 517.081,Z 538.222,A -85,B 0,C 180,E1 -5049.979,E2 -5049.979} C_VEL
LIN {X 0,Y 517.357,Z 528.327,A -85,B 0,C 180,E1 -5050.963,E2 -5050.963} C_VEL
LIN {X 0,Y 517.703,Z 517.56,A -85,B 0,C 180,E1 -5051.824,E2 -5051.824} C_VEL
LIN {X 0,Y 517.963,Z 506.383,A -85,B 0,C 180,E1 -5052.538,E2 -5052.538} C_VEL
LIN {X 0,Y 518.257,Z 494.278,A -85,B 0,C 180,E1 -5053.129,E2 -5053.129} C_VEL
LIN {X 0,Y 518.282,Z 483.465,A -85,B 0,C 180,E1 -5053.527,E2 -5053.527} C_VEL
LIN {X 0,Y 516.316,Z 472.836,A -85,B 0,C 180,E1 -5053.881,E2 -5053.881} C_VEL
LIN {X 0,Y 516.315,Z 469.795,A -85,B 0,C 180,E1 -5056.609,E2 -5056.609} C_VEL
LIN {X 0,Y 516.325,Z 466.978,A -85,B 0,C 180,E1 -5059.067,E2 -5059.067} C_VEL
LIN {X 0,Y 516.36,Z 463.284,A -85,B 0,C 180,E1 -5062.252,E2 -5062.252} C_VEL
LIN {X 0,Y 516.37,Z 459.971,A -85,B 0,C 180,E1 -5064.956,E2 -5064.956} C_VEL
LIN {X 0,Y 516.374,Z 456.499,A -85,B 0,C 180,E1 -5067.565,E2 -5067.565} C_VEL
LIN {X 0,Y 516.323,Z 452.777,A -85,B 0,C 180,E1 -5070.24,E2 -5070.24} C_VEL
LIN {X 0,Y 516.415,Z 452.162,A -85,B 0,C 180,E1 -5071.141,E2 -5071.141} C_VEL
LIN {X 0,Y 516.768,Z 452.118,A -85,B 0,C 180,E1 -5073.942,E2 -5073.942} C_VEL
LIN {X 0,Y 516.879,Z 452.103,A -85,B 0,C 180,E1 -5076.746,E2 -5076.746} C_VEL
LIN {X 0,Y 516.884,Z 452.102,A -85,B 0,C 180,E1 -5079.721,E2 -5079.721} C_VEL
LIN {X 0,Y 516.909,Z 452.098,A -85,B 0,C 180,E1 -5082.76,E2 -5082.76} C_VEL
LIN {X 0,Y 516.925,Z 452.096,A -85,B 0,C 180,E1 -5085.01,E2 -5085.01} C_VEL
LIN {X 0,Y 516.918,Z 452.099,A -85,B 0,C 180,E1 -5088.398,E2 -5088.398} C_VEL
LIN {X 0,Y 516.906,Z 452.247,A -85,B 0,C 180,E1 -5091.286,E2 -5091.286} C_VEL
LIN {X 0,Y 518.023,Z 458.688,A -85,B 0,C 180,E1 -5093.831,E2 -5093.831} C_VEL
LIN {X 0,Y 518.065,Z 464.14,A -85,B 0,C 180,E1 -5095.845,E2 -5095.845} C_VEL
LIN {X 0,Y 517.746,Z 472.909,A -85,B 0,C 180,E1 -5098.948,E2 -5098.948} C_VEL
LIN {X 0,Y 517.473,Z 481.83,A -85,B 0,C 180,E1 -5101.981,E2 -5101.981} C_VEL
LIN {X 0,Y 517.198,Z 491.292,A -85,B 0,C 180,E1 -5105.087,E2 -5105.087} C_VEL
LIN {X 0,Y 516.927,Z 501.924,A -85,B 0,C 180,E1 -5108.464,E2 -5108.464} C_VEL
LIN {X 0,Y 516.772,Z 511.335,A -85,B 0,C 180,E1 -5111.361,E2 -5111.361} C_VEL
LIN {X 0,Y 516.647,Z 520.822,A -85,B 0,C 180,E1 -5114.213,E2 -5114.213} C_VEL
LIN {X 0,Y 516.586,Z 527.092,A -85,B 0,C 180,E1 -5116.101,E2 -5116.101} C_VEL
LIN {X 0,Y 518.449,Z 540.205,A -85,B 0,C 180,E1 -5116.452,E2 -5116.452} C_VEL
LIN {X 0,Y 518.193,Z 553.331,A -85,B 0,C 180,E1 -5116.919,E2 -5116.919} C_VEL
LIN {X 0,Y 517.921,Z 565.656,A -85,B 0,C 180,E1 -5117.526,E2 -5117.526} C_VEL
LIN {X 0,Y 517.609,Z 577.004,A -85,B 0,C 180,E1 -5118.248,E2 -5118.248} C_VEL
LIN {X 0,Y 517.299,Z 588.002,A -85,B 0,C 180,E1 -5119.134,E2 -5119.134} C_VEL
LIN {X 0,Y 517.018,Z 596.962,A -85,B 0,C 180,E1 -5120.019,E2 -5120.019} C_VEL
LIN {X 0,Y 516.772,Z 606.701,A -85,B 0,C 180,E1 -5121.199,E2 -5121.199} C_VEL
LIN {X 0,Y 516.563,Z 614.455,A -85,B 0,C 180,E1 -5122.377,E2 -5122.377} C_VEL
LIN {X 0,Y 516.427,Z 621.6,A -85,B 0,C 180,E1 -5123.75,E2 -5123.75} C_VEL
LIN {X 0,Y 516.314,Z 626.349,A -85,B 0,C 180,E1 -5124.924,E2 -5124.924} C_VEL
LIN {X 0,Y 516.354,Z 629.957,A -85,B 0,C 180,E1 -5126.098,E2 -5126.098} C_VEL
LIN {X 0,Y 516.282,Z 631.806,A -85,B 0,C 180,E1 -5126.879,E2 -5126.879} C_VEL
LIN {X 0,Y 516.26,Z 633.192,A -85,B 0,C 180,E1 -5127.659,E2 -5127.659} C_VEL
LIN {X 0,Y 516.16,Z 634.785,A -85,B 0,C 180,E1 -5129.22,E2 -5129.22} C_VEL
LIN {X 0,Y 516.154,Z 635,A -85,B 0,C 180,E1 -5130,E2 -5130} C_VEL
LIN {X 0,Y 516.192,Z 634.183,A -85,B 0,C 180,E1 -5131.56,E2 -5131.56} C_VEL
LIN {X 0,Y 516.26,Z 633.195,A -85,B 0,C 180,E1 -5132.341,E2 -5132.341} C_VEL
LIN {X 0,Y 516.282,Z 631.81,A -85,B 0,C 180,E1 -5133.121,E2 -5133.121} C_VEL
LIN {X 0,Y 516.343,Z 628.891,A -85,B 0,C 180,E1 -5134.293,E2 -5134.293} C_VEL
LIN {X 0,Y 516.405,Z 624.912,A -85,B 0,C 180,E1 -5135.467,E2 -5135.467} C_VEL
LIN {X 0,Y 516.479,Z 618.962,A -85,B 0,C 180,E1 -5136.797,E2 -5136.797} C_VEL
LIN {X 0,Y 516.641,Z 612.012,A -85,B 0,C 180,E1 -5138.015,E2 -5138.015} C_VEL
LIN {X 0,Y 516.844,Z 603.644,A -85,B 0,C 180,E1 -5139.194,E2 -5139.194} C_VEL
LIN {X 0,Y 517.058,Z 595.054,A -85,B 0,C 180,E1 -5140.178,E2 -5140.178} C_VEL
LIN {X 0,Y 517.416,Z 584.449,A -85,B 0,C 180,E1 -5141.16,E2 -5141.16} C_VEL
LIN {X 0,Y 517.697,Z 572.573,A -85,B 0,C 180,E1 -5142.043,E2 -5142.043} C_VEL
LIN {X 0,Y 518.007,Z 560.478,A -85,B 0,C 180,E1 -5142.737,E2 -5142.737} C_VEL
LIN {X 0,Y 518.274,Z 547.992,A -85,B 0,C 180,E1 -5143.278,E2 -5143.278} C_VEL
LIN {X 0,Y 518.221,Z 537.917,A -85,B 0,C 180,E1 -5143.604,E2 -5143.604} C_VEL
LIN {X 0,Y 516.569,Z 526.747,A -85,B 0,C 180,E1 -5143.899,E2 -5143.899} C_VEL
LIN {X 0,Y 516.623,Z 517.508,A -85,B 0,C 180,E1 -5146.599,E2 -5146.599} C_VEL
LIN {X 0,Y 516.753,Z 507.736,A -85,B 0,C 180,E1 -5149.464,E2 -5149.464} C_VEL
LIN {X 0,Y 516.902,Z 498.048,A -85,B 0,C 180,E1 -5152.398,E2 -5152.398} C_VEL
LIN {X 0,Y 517.067,Z 488.592,A -85,B 0,C 180,E1 -5155.35,E2 -5155.35} C_VEL
LIN {X 0,Y 517.247,Z 480.585,A -85,B 0,C 180,E1 -5157.972,E2 -5157.972} C_VEL
LIN {X 0,Y 517.581,Z 471.426,A -85,B 0,C 180,E1 -5161.19,E2 -5161.19} C_VEL
LIN {X 0,Y 517.951,Z 463.912,A -85,B 0,C 180,E1 -5164.137,E2 -5164.137} C_VEL
LIN {X 0,Y 518.131,Z 460.415,A -85,B 0,C 180,E1 -5165.68,E2 -5165.68} C_VEL
LIN {X 0,Y 517.729,Z 456.633,A -85,B 0,C 180,E1 -5167.652,E2 -5167.652} C_VEL
LIN {X 0,Y 517.138,Z 453.466,A -85,B 0,C 180,E1 -5169.698,E2 -5169.698} C_VEL
LIN {X 0,Y 516.906,Z 452.169,A -85,B 0,C 180,E1 -5170.74,E2 -5170.74} C_VEL
LIN {X 0,Y 516.885,Z 452.103,A -85,B 0,C 180,E1 -5173.903,E2 -5173.903} C_VEL
LIN {X 0,Y 516.885,Z 452.103,A -85,B 0,C 180,E1 -5176.107,E2 -5176.107} C_VEL
LIN {X 0,Y 516.92,Z 452.099,A -85,B 0,C 180,E1 -5178.398,E2 -5178.398} C_VEL
LIN {X 0,Y 516.886,Z 452.103,A -85,B 0,C 180,E1 -5181.284,E2 -5181.284} C_VEL
LIN {X 0,Y 516.849,Z 452.296,A -85,B 0,C 180,E1 -5184.218,E2 -5184.218} C_VEL
LIN {X 0,Y 516.898,Z 453.753,A -85,B 0,C 180,E1 -5186.12,E2 -5186.12} C_VEL
LIN {X 0,Y 516.776,Z 456.139,A -85,B 0,C 180,E1 -5188.958,E2 -5188.958} C_VEL
LIN {X 0,Y 516.644,Z 458.463,A -85,B 0,C 180,E1 -5191.568,E2 -5191.568} C_VEL
LIN {X 0,Y 516.58,Z 460.901,A -85,B 0,C 180,E1 -5194.192,E2 -5194.192} C_VEL
LIN {X 0,Y 516.473,Z 463.37,A -85,B 0,C 180,E1 -5196.758,E2 -5196.758} C_VEL
LIN {X 0,Y 516.437,Z 466.473,A -85,B 0,C 180,E1 -5199.884,E2 -5199.884} C_VEL
LIN {X 0,Y 516.37,Z 469.198,A -85,B 0,C 180,E1 -5202.577,E2 -5202.577} C_VEL
LIN {X 0,Y 516.369,Z 471.797,A -85,B 0,C 180,E1 -5205.093,E2 -5205.093} C_VEL
LIN {X 0,Y 516.313,Z 473.008,A -85,B 0,C 180,E1 -5206.219,E2 -5206.219} C_VEL
LIN {X 0,Y 518.452,Z 484.731,A -85,B 0,C 180,E1 -5206.602,E2 -5206.602} C_VEL
LIN {X 0,Y 518.175,Z 497.984,A -85,B 0,C 180,E1 -5207.118,E2 -5207.118} C_VEL
LIN {X 0,Y 517.879,Z 510.472,A -85,B 0,C 180,E1 -5207.789,E2 -5207.789} C_VEL
LIN {X 0,Y 517.612,Z 521.398,A -85,B 0,C 180,E1 -5208.547,E2 -5208.547} C_VEL
LIN {X 0,Y 517.289,Z 531.681,A -85,B 0,C 180,E1 -5209.431,E2 -5209.431} C_VEL
LIN {X 0,Y 517.006,Z 540.914,A -85,B 0,C 180,E1 -5210.414,E2 -5210.414} C_VEL
LIN {X 0,Y 516.778,Z 549.836,A -85,B 0,C 180,E1 -5211.594,E2 -5211.594} C_VEL
LIN {X 0,Y 516.576,Z 557.015,A -85,B 0,C 180,E1 -5212.771,E2 -5212.771} C_VEL
LIN {X 0,Y 516.474,Z 561.855,A -85,B 0,C 180,E1 -5213.75,E2 -5213.75} C_VEL
LIN {X 0,Y 516.313,Z 566.555,A -85,B 0,C 180,E1 -5214.924,E2 -5214.924} C_VEL
LIN {X 0,Y 516.373,Z 570.142,A -85,B 0,C 180,E1 -5216.098,E2 -5216.098} C_VEL
LIN {X 0,Y 516.283,Z 572.001,A -85,B 0,C 180,E1 -5216.879,E2 -5216.879} C_VEL
LIN {X 0,Y 516.261,Z 573.402,A -85,B 0,C 180,E1 -5217.66,E2 -5217.66} C_VEL
LIN {X 0,Y 516.16,Z 575.012,A -85,B 0,C 180,E1 -5219.22,E2 -5219.22} C_VEL
LIN {X 0,Y 516.154,Z 575.245,A -85,B 0,C 180,E1 -5220,E2 -5220} C_VEL
LIN {X 0,Y 516.16,Z 575.06,A -85,B 0,C 180,E1 -5220.78,E2 -5220.78} C_VEL
LIN {X 0,Y 516.26,Z 573.512,A -85,B 0,C 180,E1 -5222.341,E2 -5222.341} C_VEL
LIN {X 0,Y 516.283,Z 572.159,A -85,B 0,C 180,E1 -5223.122,E2 -5223.122} C_VEL
LIN {X 0,Y 516.361,Z 569.301,A -85,B 0,C 180,E1 -5224.293,E2 -5224.293} C_VEL
LIN {X 0,Y 516.4,Z 565.426,A -85,B 0,C 180,E1 -5225.467,E2 -5225.467} C_VEL
LIN {X 0,Y 516.491,Z 559.555,A -85,B 0,C 180,E1 -5226.817,E2 -5226.817} C_VEL
LIN {X 0,Y 516.647,Z 552.886,A -85,B 0,C 180,E1 -5228.015,E2 -5228.015} C_VEL
LIN {X 0,Y 516.846,Z 544.723,A -85,B 0,C 180,E1 -5229.194,E2 -5229.194} C_VEL
LIN {X 0,Y 517.101,Z 536.354,A -85,B 0,C 180,E1 -5230.177,E2 -5230.177} C_VEL
LIN {X 0,Y 517.455,Z 526.003,A -85,B 0,C 180,E1 -5231.16,E2 -5231.16} C_VEL
LIN {X 0,Y 517.737,Z 514.503,A -85,B 0,C 180,E1 -5232.035,E2 -5232.035} C_VEL
LIN {X 0,Y 518.023,Z 502.686,A -85,B 0,C 180,E1 -5232.737,E2 -5232.737} C_VEL
LIN {X 0,Y 518.302,Z 490.589,A -85,B 0,C 180,E1 -5233.278,E2 -5233.278} C_VEL
LIN {X 0,Y 518.282,Z 483.547,A -85,B 0,C 180,E1 -5233.528,E2 -5233.528} C_VEL
LIN {X 0,Y 516.317,Z 472.472,A -85,B 0,C 180,E1 -5233.881,E2 -5233.881} C_VEL
LIN {X 0,Y 516.278,Z 469.363,A -85,B 0,C 180,E1 -5236.611,E2 -5236.611} C_VEL
LIN {X 0,Y 516.319,Z 466.646,A -85,B 0,C 180,E1 -5239.068,E2 -5239.068} C_VEL
LIN {X 0,Y 516.328,Z 463.854,A -85,B 0,C 180,E1 -5241.563,E2 -5241.563} C_VEL
LIN {X 0,Y 516.381,Z 460.895,A -85,B 0,C 180,E1 -5244.233,E2 -5244.233} C_VEL
LIN {X 0,Y 516.431,Z 458.191,A -85,B 0,C 180,E1 -5246.686,E2 -5246.686} C_VEL
LIN {X 0,Y 516.47,Z 455.166,A -85,B 0,C 180,E1 -5249.437,E2 -5249.437} C_VEL
LIN {X 0,Y 516.478,Z 452.325,A -85,B 0,C 180,E1 -5252.053,E2 -5252.053} C_VEL
LIN {X 0,Y 516.805,Z 452.113,A -85,B 0,C 180,E1 -5254.831,E2 -5254.831} C_VEL
LIN {X 0,Y 516.884,Z 452.098,A -85,B 0,C 180,E1 -5257.943,E2 -5257.943} C_VEL
LIN {X 0,Y 516.889,Z 452.098,A -85,B 0,C 180,E1 -5260.742,E2 -5260.742} C_VEL
LIN {X 0,Y 516.902,Z 452.095,A -85,B 0,C 180,E1 -5262.906,E2 -5262.906} C_VEL
LIN {X 0,Y 516.928,Z 452.093,A -85,B 0,C 180,E1 -5265.01,E2 -5265.01} C_VEL
LIN {X 0,Y 516.873,Z 452.099,A -85,B 0,C 180,E1 -5266.305,E2 -5266.305} C_VEL
LIN {X 0,Y 516.197,Z 452.187,A -85,B 0,C 180,E1 -5266.956,E2 -5266.956} C_VEL
LIN {X 0,Y 513.362,Z 452.537,A -85,B 0,C 180,E1 -5268.013,E2 -5268.013} C_VEL
LIN {X 0,Y 510.966,Z 452.84,A -85,B 0,C 180,E1 -5268.865,E2 -5268.865} C_VEL
LIN {X 0,Y 509.926,Z 452.966,A -85,B 0,C 180,E1 -5269.522,E2 -5269.522} C_VEL
LIN {X 0,Y 509.834,Z 452.976,A -85,B 0,C 180,E1 -5269.745,E2 -5269.745} C_VEL
LIN {X 0,Y 509.821,Z 452.98,A -85,B 0,C 180,E1 -5272.659,E2 -5272.659} C_VEL
LIN {X 0,Y 509.862,Z 452.977,A -85,B 0,C 180,E1 -5275.797,E2 -5275.797} C_VEL
LIN {X 0,Y 509.851,Z 452.975,A -85,B 0,C 180,E1 -5278.72,E2 -5278.72} C_VEL
LIN {X 0,Y 509.902,Z 452.968,A -85,B 0,C 180,E1 -5281.9,E2 -5281.9} C_VEL
LIN {X 0,Y 509.846,Z 452.976,A -85,B 0,C 180,E1 -5284.702,E2 -5284.702} C_VEL
LIN {X 0,Y 509.832,Z 452.977,A -85,B 0,C 180,E1 -5287.458,E2 -5287.458} C_VEL
LIN {X 0,Y 509.923,Z 452.969,A -85,B 0,C 180,E1 -5289.845,E2 -5289.845} C_VEL
LIN {X 0,Y 509.88,Z 452.974,A -85,B 0,C 180,E1 -5293.174,E2 -5293.174} C_VEL
LIN {X 0,Y 509.87,Z 452.972,A -85,B 0,C 180,E1 -5295.634,E2 -5295.634} C_VEL
LIN {X 0,Y 509.919,Z 452.964,A -85,B 0,C 180,E1 -5298.875,E2 -5298.875} C_VEL
LIN {X 0,Y 509.957,Z 452.962,A -85,B 0,C 180,E1 -5302.079,E2 -5302.079} C_VEL
LIN {X 0,Y 509.985,Z 452.958,A -85,B 0,C 180,E1 -5304.464,E2 -5304.464} C_VEL
LIN {X 0,Y 510.061,Z 452.948,A -85,B 0,C 180,E1 -5307.631,E2 -5307.631} C_VEL
LIN {X 0,Y 510.069,Z 452.946,A -85,B 0,C 180,E1 -5310.789,E2 -5310.789} C_VEL
LIN {X 0,Y 509.959,Z 452.961,A -85,B 0,C 180,E1 -5313.16,E2 -5313.16} C_VEL
LIN {X 0,Y 509.943,Z 452.963,A -85,B 0,C 180,E1 -5316.33,E2 -5316.33} C_VEL
LIN {X 0,Y 509.91,Z 452.971,A -85,B 0,C 180,E1 -5318.72,E2 -5318.72} C_VEL
LIN {X 0,Y 509.911,Z 452.97,A -85,B 0,C 180,E1 -5321.932,E2 -5321.932} C_VEL
LIN {X 0,Y 509.9,Z 452.969,A -85,B 0,C 180,E1 -5325.242,E2 -5325.242} C_VEL
LIN {X 0,Y 509.888,Z 452.97,A -85,B 0,C 180,E1 -5327.998,E2 -5327.998} C_VEL
LIN {X 0,Y 509.856,Z 452.977,A -85,B 0,C 180,E1 -5331.002,E2 -5331.002} C_VEL
LIN {X 0,Y 509.828,Z 452.977,A -85,B 0,C 180,E1 -5333.564,E2 -5333.564} C_VEL
LIN {X 0,Y 509.916,Z 452.966,A -85,B 0,C 180,E1 -5336.378,E2 -5336.378} C_VEL
LIN {X 0,Y 509.882,Z 452.971,A -85,B 0,C 180,E1 -5338.844,E2 -5338.844} C_VEL
LIN {X 0,Y 509.825,Z 452.979,A -85,B 0,C 180,E1 -5341.59,E2 -5341.59} C_VEL
LIN {X 0,Y 509.857,Z 452.978,A -85,B 0,C 180,E1 -5344.413,E2 -5344.413} C_VEL
LIN {X 0,Y 509.823,Z 452.977,A -85,B 0,C 180,E1 -5347.34,E2 -5347.34} C_VEL
LIN {X 0,Y 509.843,Z 452.974,A -85,B 0,C 180,E1 -5350.382,E2 -5350.382} C_VEL
LIN {X 0,Y 509.827,Z 452.981,A -85,B 0,C 180,E1 -5353.062,E2 -5353.062} C_VEL
LIN {X 0,Y 509.835,Z 452.977,A -85,B 0,C 180,E1 -5355.792,E2 -5355.792} C_VEL
LIN {X 0,Y 509.862,Z 452.975,A -85,B 0,C 180,E1 -5358.575,E2 -5358.575} C_VEL
LIN {X 0,Y 509.855,Z 452.978,A -85,B 0,C 180,E1 -5361.786,E2 -5361.786} C_VEL
LIN {X 0,Y 509.792,Z 452.982,A -85,B 0,C 180,E1 -5364.618,E2 -5364.618} C_VEL
LIN {X 0,Y 509.554,Z 453.017,A -85,B 0,C 180,E1 -5367.458,E2 -5367.458} C_VEL
LIN {X 0,Y 509.36,Z 453.041,A -85,B 0,C 180,E1 -5368.811,E2 -5368.811} C_VEL
LIN {X 0,Y 509.305,Z 454.62,A -85,B 0,C 180,E1 -5370.384,E2 -5370.384} C_VEL
LIN {X 0,Y 509.34,Z 457.616,A -85,B 0,C 180,E1 -5372.913,E2 -5372.913} C_VEL
LIN {X 0,Y 509.303,Z 460.749,A -85,B 0,C 180,E1 -5375.61,E2 -5375.61} C_VEL
LIN {X 0,Y 509.247,Z 463.671,A -85,B 0,C 180,E1 -5378.122,E2 -5378.122} C_VEL
LIN {X 0,Y 509.228,Z 466.594,A -85,B 0,C 180,E1 -5380.656,E2 -5380.656} C_VEL
LIN {X 0,Y 509.204,Z 469.474,A -85,B 0,C 180,E1 -5383.151,E2 -5383.151} C_VEL
LIN {X 0,Y 509.256,Z 472.969,A -85,B 0,C 180,E1 -5386.037,E2 -5386.037} C_VEL
LIN {X 0,Y 511.532,Z 485.411,A -85,B 0,C 180,E1 -5386.442,E2 -5386.442} C_VEL
LIN {X 0,Y 511.248,Z 497.87,A -85,B 0,C 180,E1 -5386.94,E2 -5386.94} C_VEL
LIN {X 0,Y 510.975,Z 509.569,A -85,B 0,C 180,E1 -5387.566,E2 -5387.566} C_VEL
LIN {X 0,Y 510.685,Z 520.168,A -85,B 0,C 180,E1 -5388.288,E2 -5388.288} C_VEL
LIN {X 0,Y 510.327,Z 530.686,A -85,B 0,C 180,E1 -5389.185,E2 -5389.185} C_VEL
LIN {X 0,Y 510.006,Z 541.036,A -85,B 0,C 180,E1 -5390.281,E2 -5390.281} C_VEL
LIN {X 0,Y 509.717,Z 550.02,A -85,B 0,C 180,E1 -5391.476,E2 -5391.476} C_VEL
LIN {X 0,Y 509.495,Z 557.23,A -85,B 0,C 180,E1 -5392.669,E2 -5392.669} C_VEL
LIN {X 0,Y 509.388,Z 562.12,A -85,B 0,C 180,E1 -5393.663,E2 -5393.663} C_VEL
LIN {X 0,Y 509.251,Z 566.853,A -85,B 0,C 180,E1 -5394.853,E2 -5394.853} C_VEL
LIN {X 0,Y 509.304,Z 570.47,A -85,B 0,C 180,E1 -5396.043,E2 -5396.043} C_VEL
LIN {X 0,Y 509.202,Z 572.323,A -85,B 0,C 180,E1 -5396.835,E2 -5396.835} C_VEL
LIN {X 0,Y 509.189,Z 573.741,A -85,B 0,C 180,E1 -5397.627,E2 -5397.627} C_VEL
LIN {X 0,Y 509.112,Z 574.77,A -85,B 0,C 180,E1 -5398.418,E2 -5398.418} C_VEL
LIN {X 0,Y 509.074,Z 575.389,A -85,B 0,C 180,E1 -5399.209,E2 -5399.209} C_VEL
LIN {X 0,Y 509.074,Z 575.451,A -85,B 0,C 180,E1 -5400.791,E2 -5400.791} C_VEL
LIN {X 0,Y 509.113,Z 574.883,A -85,B 0,C 180,E1 -5401.582,E2 -5401.582} C_VEL
LIN {X 0,Y 509.216,Z 572.563,A -85,B 0,C 180,E1 -5403.165,E2 -5403.165} C_VEL
LIN {X 0,Y 509.283,Z 569.716,A -85,B 0,C 180,E1 -5404.353,E2 -5404.353} C_VEL
LIN {X 0,Y 509.341,Z 565.841,A -85,B 0,C 180,E1 -5405.543,E2 -5405.543} C_VEL
LIN {X 0,Y 509.448,Z 560.095,A -85,B 0,C 180,E1 -5406.882,E2 -5406.882} C_VEL
LIN {X 0,Y 509.631,Z 553.281,A -85,B 0,C 180,E1 -5408.126,E2 -5408.126} C_VEL
LIN {X 0,Y 509.843,Z 545.11,A -85,B 0,C 180,E1 -5409.321,E2 -5409.321} C_VEL
LIN {X 0,Y 510.121,Z 536.683,A -85,B 0,C 180,E1 -5410.317,E2 -5410.317} C_VEL
LIN {X 0,Y 510.496,Z 526.331,A -85,B 0,C 180,E1 -5411.314,E2 -5411.314} C_VEL
LIN {X 0,Y 510.858,Z 515.163,A -85,B 0,C 180,E1 -5412.172,E2 -5412.172} C_VEL
LIN {X 0,Y 511.093,Z 504.718,A -85,B 0,C 180,E1 -5412.811,E2 -5412.811} C_VEL
LIN {X 0,Y 511.393,Z 491.99,A -85,B 0,C 180,E1 -5413.409,E2 -5413.409} C_VEL
LIN {X 0,Y 511.326,Z 483.907,A -85,B 0,C 180,E1 -5413.702,E2 -5413.702} C_VEL
LIN {X 0,Y 509.269,Z 473.357,A -85,B 0,C 180,E1 -5414.052,E2 -5414.052} C_VEL
LIN {X 0,Y 509.301,Z 469.226,A -85,B 0,C 180,E1 -5417.673,E2 -5417.673} C_VEL
LIN {X 0,Y 509.303,Z 466.263,A -85,B 0,C 180,E1 -5420.223,E2 -5420.223} C_VEL
LIN {X 0,Y 509.263,Z 463.271,A -85,B 0,C 180,E1 -5422.731,E2 -5422.731} C_VEL
LIN {X 0,Y 509.314,Z 460.068,A -85,B 0,C 180,E1 -5425.326,E2 -5425.326} C_VEL
LIN {X 0,Y 509.289,Z 456.559,A -85,B 0,C 180,E1 -5427.982,E2 -5427.982} C_VEL
LIN {X 0,Y 509.29,Z 453.05,A -85,B 0,C 180,E1 -5430.703,E2 -5430.703} C_VEL
LIN {X 0,Y 509.669,Z 453.002,A -85,B 0,C 180,E1 -5433.475,E2 -5433.475} C_VEL
LIN {X 0,Y 509.814,Z 452.981,A -85,B 0,C 180,E1 -5436.354,E2 -5436.354} C_VEL
LIN {X 0,Y 509.848,Z 452.978,A -85,B 0,C 180,E1 -5439.352,E2 -5439.352} C_VEL
LIN {X 0,Y 509.851,Z 452.977,A -85,B 0,C 180,E1 -5442.488,E2 -5442.488} C_VEL
LIN {X 0,Y 509.859,Z 452.976,A -85,B 0,C 180,E1 -5445.332,E2 -5445.332} C_VEL
LIN {X 0,Y 509.859,Z 452.978,A -85,B 0,C 180,E1 -5448.575,E2 -5448.575} C_VEL
LIN {X 0,Y 509.886,Z 453.131,A -85,B 0,C 180,E1 -5451.033,E2 -5451.033} C_VEL
LIN {X 0,Y 511.048,Z 459.884,A -85,B 0,C 180,E1 -5453.748,E2 -5453.748} C_VEL
LIN {X 0,Y 511.113,Z 464.798,A -85,B 0,C 180,E1 -5455.591,E2 -5455.591} C_VEL
LIN {X 0,Y 510.797,Z 472.998,A -85,B 0,C 180,E1 -5458.545,E2 -5458.545} C_VEL
LIN {X 0,Y 510.471,Z 480.631,A -85,B 0,C 180,E1 -5461.192,E2 -5461.192} C_VEL
LIN {X 0,Y 510.256,Z 488.494,A -85,B 0,C 180,E1 -5463.848,E2 -5463.848} C_VEL
LIN {X 0,Y 509.968,Z 497.739,A -85,B 0,C 180,E1 -5466.873,E2 -5466.873} C_VEL
LIN {X 0,Y 509.774,Z 507.045,A -85,B 0,C 180,E1 -5469.839,E2 -5469.839} C_VEL
LIN {X 0,Y 509.63,Z 516.437,A -85,B 0,C 180,E1 -5472.753,E2 -5472.753} C_VEL
LIN {X 0,Y 509.494,Z 526.489,A -85,B 0,C 180,E1 -5475.827,E2 -5475.827} C_VEL
LIN {X 0,Y 509.481,Z 526.739,A -85,B 0,C 180,E1 -5475.903,E2 -5475.903} C_VEL
LIN {X 0,Y 511.516,Z 540.489,A -85,B 0,C 180,E1 -5476.29,E2 -5476.29} C_VEL
LIN {X 0,Y 511.266,Z 552.792,A -85,B 0,C 180,E1 -5476.739,E2 -5476.739} C_VEL
LIN {X 0,Y 510.964,Z 565.307,A -85,B 0,C 180,E1 -5477.364,E2 -5477.364} C_VEL
LIN {X 0,Y 510.616,Z 576.487,A -85,B 0,C 180,E1 -5478.085,E2 -5478.085} C_VEL
LIN {X 0,Y 510.29,Z 587.513,A -85,B 0,C 180,E1 -5478.983,E2 -5478.983} C_VEL
LIN {X 0,Y 509.979,Z 596.488,A -85,B 0,C 180,E1 -5479.88,E2 -5479.88} C_VEL
LIN {X 0,Y 509.712,Z 606.241,A -85,B 0,C 180,E1 -5481.076,E2 -5481.076} C_VEL
LIN {X 0,Y 509.494,Z 614.015,A -85,B 0,C 180,E1 -5482.271,E2 -5482.271} C_VEL
LIN {X 0,Y 509.326,Z 621.171,A -85,B 0,C 180,E1 -5483.662,E2 -5483.662} C_VEL
LIN {X 0,Y 509.248,Z 625.934,A -85,B 0,C 180,E1 -5484.853,E2 -5484.853} C_VEL
LIN {X 0,Y 509.268,Z 629.576,A -85,B 0,C 180,E1 -5486.043,E2 -5486.043} C_VEL
LIN {X 0,Y 509.2,Z 631.449,A -85,B 0,C 180,E1 -5486.835,E2 -5486.835} C_VEL
LIN {X 0,Y 509.189,Z 632.856,A -85,B 0,C 180,E1 -5487.627,E2 -5487.627} C_VEL
LIN {X 0,Y 509.073,Z 634.465,A -85,B 0,C 180,E1 -5489.209,E2 -5489.209} C_VEL
LIN {X 0,Y 509.065,Z 634.679,A -85,B 0,C 180,E1 -5490,E2 -5490} C_VEL
LIN {X 0,Y 509.112,Z 633.848,A -85,B 0,C 180,E1 -5491.582,E2 -5491.582} C_VEL
LIN {X 0,Y 509.189,Z 632.846,A -85,B 0,C 180,E1 -5492.373,E2 -5492.373} C_VEL
LIN {X 0,Y 509.2,Z 631.43,A -85,B 0,C 180,E1 -5493.165,E2 -5493.165} C_VEL
LIN {X 0,Y 509.232,Z 628.46,A -85,B 0,C 180,E1 -5494.353,E2 -5494.353} C_VEL
LIN {X 0,Y 509.322,Z 624.44,A -85,B 0,C 180,E1 -5495.543,E2 -5495.543} C_VEL
LIN {X 0,Y 509.402,Z 618.705,A -85,B 0,C 180,E1 -5496.844,E2 -5496.844} C_VEL
LIN {X 0,Y 509.573,Z 611.48,A -85,B 0,C 180,E1 -5498.127,E2 -5498.127} C_VEL
LIN {X 0,Y 509.782,Z 603.073,A -85,B 0,C 180,E1 -5499.322,E2 -5499.322} C_VEL
LIN {X 0,Y 510.031,Z 594.443,A -85,B 0,C 180,E1 -5500.319,E2 -5500.319} C_VEL
LIN {X 0,Y 510.388,Z 583.796,A -85,B 0,C 180,E1 -5501.316,E2 -5501.316} C_VEL
LIN {X 0,Y 510.694,Z 571.875,A -85,B 0,C 180,E1 -5502.211,E2 -5502.211} C_VEL
LIN {X 0,Y 511.033,Z 559.725,A -85,B 0,C 180,E1 -5502.913,E2 -5502.913} C_VEL
LIN {X 0,Y 511.301,Z 547.225,A -85,B 0,C 180,E1 -5503.463,E2 -5503.463} C_VEL
LIN {X 0,Y 511.284,Z 538.914,A -85,B 0,C 180,E1 -5503.742,E2 -5503.742} C_VEL
LIN {X 0,Y 509.474,Z 526.221,A -85,B 0,C 180,E1 -5504.097,E2 -5504.097} C_VEL
LIN {X 0,Y 509.554,Z 517.029,A -85,B 0,C 180,E1 -5506.837,E2 -5506.837} C_VEL
LIN {X 0,Y 509.683,Z 507.317,A -85,B 0,C 180,E1 -5509.745,E2 -5509.745} C_VEL
LIN {X 0,Y 509.858,Z 497.712,A -85,B 0,C 180,E1 -5512.703,E2 -5512.703} C_VEL
LIN {X 0,Y 510.075,Z 488.276,A -85,B 0,C 180,E1 -5515.723,E2 -5515.723} C_VEL
LIN {X 0,Y 510.223,Z 481.001,A -85,B 0,C 180,E1 -5518.169,E2 -5518.169} C_VEL
LIN {X 0,Y 510.562,Z 473.08,A -85,B 0,C 180,E1 -5521.018,E2 -5521.018} C_VEL
LIN {X 0,Y 510.963,Z 465.954,A -85,B 0,C 180,E1 -5523.852,E2 -5523.852} C_VEL
LIN {X 0,Y 511.166,Z 461.649,A -85,B 0,C 180,E1 -5525.788,E2 -5525.788} C_VEL
LIN {X 0,Y 510.906,Z 458.858,A -85,B 0,C 180,E1 -5527.248,E2 -5527.248} C_VEL
LIN {X 0,Y 510.271,Z 455.297,A -85,B 0,C 180,E1 -5529.53,E2 -5529.53} C_VEL
LIN {X 0,Y 509.869,Z 453.055,A -85,B 0,C 180,E1 -5531.424,E2 -5531.424} C_VEL
LIN {X 0,Y 509.859,Z 452.978,A -85,B 0,C 180,E1 -5534.668,E2 -5534.668} C_VEL
LIN {X 0,Y 509.864,Z 452.977,A -85,B 0,C 180,E1 -5538.103,E2 -5538.103} C_VEL
LIN {X 0,Y 509.85,Z 452.979,A -85,B 0,C 180,E1 -5540.648,E2 -5540.648} C_VEL
LIN {X 0,Y 509.801,Z 453.046,A -85,B 0,C 180,E1 -5543.645,E2 -5543.645} C_VEL
LIN {X 0,Y 509.83,Z 455.143,A -85,B 0,C 180,E1 -5546.537,E2 -5546.537} C_VEL
LIN {X 0,Y 509.725,Z 457.43,A -85,B 0,C 180,E1 -5549.326,E2 -5549.326} C_VEL
LIN {X 0,Y 509.595,Z 459.802,A -85,B 0,C 180,E1 -5552.037,E2 -5552.037} C_VEL
LIN {X 0,Y 509.511,Z 462.229,A -85,B 0,C 180,E1 -5554.685,E2 -5554.685} C_VEL
LIN {X 0,Y 509.409,Z 464.963,A -85,B 0,C 180,E1 -5557.572,E2 -5557.572} C_VEL
LIN {X 0,Y 509.325,Z 468.019,A -85,B 0,C 180,E1 -5560.66,E2 -5560.66} C_VEL
LIN {X 0,Y 509.289,Z 470.549,A -85,B 0,C 180,E1 -5563.155,E2 -5563.155} C_VEL
LIN {X 0,Y 509.295,Z 473.097,A -85,B 0,C 180,E1 -5565.618,E2 -5565.618} C_VEL
LIN {X 0,Y 509.262,Z 473.531,A -85,B 0,C 180,E1 -5566.025,E2 -5566.025} C_VEL
LIN {X 0,Y 511.533,Z 485.645,A -85,B 0,C 180,E1 -5566.442,E2 -5566.442} C_VEL
LIN {X 0,Y 511.275,Z 498.186,A -85,B 0,C 180,E1 -5566.941,E2 -5566.941} C_VEL
LIN {X 0,Y 511.024,Z 509.451,A -85,B 0,C 180,E1 -5567.542,E2 -5567.542} C_VEL
LIN {X 0,Y 510.706,Z 520.4,A -85,B 0,C 180,E1 -5568.289,E2 -5568.289} C_VEL
LIN {X 0,Y 510.331,Z 530.931,A -85,B 0,C 180,E1 -5569.185,E2 -5569.185} C_VEL
LIN {X 0,Y 510.086,Z 539.533,A -85,B 0,C 180,E1 -5570.083,E2 -5570.083} C_VEL
LIN {X 0,Y 509.831,Z 547.446,A -85,B 0,C 180,E1 -5571.079,E2 -5571.079} C_VEL
LIN {X 0,Y 509.579,Z 555.187,A -85,B 0,C 180,E1 -5572.272,E2 -5572.272} C_VEL
LIN {X 0,Y 509.429,Z 562.25,A -85,B 0,C 180,E1 -5573.664,E2 -5573.664} C_VEL
LIN {X 0,Y 509.249,Z 566.961,A -85,B 0,C 180,E1 -5574.854,E2 -5574.854} C_VEL
LIN {X 0,Y 509.303,Z 570.555,A -85,B 0,C 180,E1 -5576.044,E2 -5576.044} C_VEL
LIN {X 0,Y 509.215,Z 572.416,A -85,B 0,C 180,E1 -5576.835,E2 -5576.835} C_VEL
LIN {X 0,Y 509.189,Z 573.819,A -85,B 0,C 180,E1 -5577.627,E2 -5577.627} C_VEL
LIN {X 0,Y 509.074,Z 575.428,A -85,B 0,C 180,E1 -5579.209,E2 -5579.209} C_VEL
LIN {X 0,Y 509.067,Z 575.658,A -85,B 0,C 180,E1 -5580,E2 -5580} C_VEL
LIN {X 0,Y 509.074,Z 575.469,A -85,B 0,C 180,E1 -5580.791,E2 -5580.791} C_VEL
LIN {X 0,Y 509.189,Z 573.909,A -85,B 0,C 180,E1 -5582.373,E2 -5582.373} C_VEL
LIN {X 0,Y 509.202,Z 572.546,A -85,B 0,C 180,E1 -5583.165,E2 -5583.165} C_VEL
LIN {X 0,Y 509.283,Z 569.673,A -85,B 0,C 180,E1 -5584.353,E2 -5584.353} C_VEL
LIN {X 0,Y 509.339,Z 565.78,A -85,B 0,C 180,E1 -5585.543,E2 -5585.543} C_VEL
LIN {X 0,Y 509.455,Z 560.101,A -85,B 0,C 180,E1 -5586.869,E2 -5586.869} C_VEL
LIN {X 0,Y 509.623,Z 553.193,A -85,B 0,C 180,E1 -5588.126,E2 -5588.126} C_VEL
LIN {X 0,Y 509.837,Z 545.001,A -85,B 0,C 180,E1 -5589.322,E2 -5589.322} C_VEL
LIN {X 0,Y 510.108,Z 536.605,A -85,B 0,C 180,E1 -5590.318,E2 -5590.318} C_VEL
LIN {X 0,Y 510.505,Z 526.218,A -85,B 0,C 180,E1 -5591.314,E2 -5591.314} C_VEL
LIN {X 0,Y 510.791,Z 514.694,A -85,B 0,C 180,E1 -5592.201,E2 -5592.201} C_VEL
LIN {X 0,Y 511.093,Z 502.824,A -85,B 0,C 180,E1 -5592.912,E2 -5592.912} C_VEL
LIN {X 0,Y 511.415,Z 489.431,A -85,B 0,C 180,E1 -5593.51,E2 -5593.51} C_VEL
LIN {X 0,Y 511.36,Z 484.396,A -85,B 0,C 180,E1 -5593.689,E2 -5593.689} C_VEL
LIN {X 0,Y 509.236,Z 472.826,A -85,B 0,C 180,E1 -5594.078,E2 -5594.078} C_VEL
LIN {X 0,Y 509.213,Z 469.708,A -85,B 0,C 180,E1 -5596.848,E2 -5596.848} C_VEL
LIN {X 0,Y 509.245,Z 466.92,A -85,B 0,C 180,E1 -5599.343,E2 -5599.343} C_VEL
LIN {X 0,Y 509.29,Z 463.513,A -85,B 0,C 180,E1 -5602.395,E2 -5602.395} C_VEL
LIN {X 0,Y 509.349,Z 460.309,A -85,B 0,C 180,E1 -5605.324,E2 -5605.324} C_VEL
LIN {X 0,Y 509.368,Z 457.36,A -85,B 0,C 180,E1 -5607.988,E2 -5607.988} C_VEL
LIN {X 0,Y 509.41,Z 453.892,A -85,B 0,C 180,E1 -5611.198,E2 -5611.198} C_VEL
LIN {X 0,Y 509.485,Z 453.026,A -85,B 0,C 180,E1 -5612.547,E2 -5612.547} C_VEL
LIN {X 0,Y 509.774,Z 452.987,A -85,B 0,C 180,E1 -5615.383,E2 -5615.383} C_VEL
LIN {X 0,Y 509.854,Z 452.976,A -85,B 0,C 180,E1 -5618.338,E2 -5618.338} C_VEL
LIN {X 0,Y 509.862,Z 452.971,A -85,B 0,C 180,E1 -5621.426,E2 -5621.426} C_VEL
LIN {X 0,Y 509.862,Z 452.973,A -85,B 0,C 180,E1 -5624.668,E2 -5624.668} C_VEL
LIN {X 0,Y 509.86,Z 452.973,A -85,B 0,C 180,E1 -5628.104,E2 -5628.104} C_VEL
LIN {X 0,Y 509.834,Z 452.976,A -85,B 0,C 180,E1 -5629.745,E2 -5629.745} C_VEL
LIN {X 0,Y 509.152,Z 453.065,A -85,B 0,C 180,E1 -5630.404,E2 -5630.404} C_VEL
LIN {X 0,Y 506.304,Z 453.416,A -85,B 0,C 180,E1 -5631.476,E2 -5631.476} C_VEL
LIN {X 0,Y 503.899,Z 453.721,A -85,B 0,C 180,E1 -5632.339,E2 -5632.339} C_VEL
LIN {X 0,Y 502.857,Z 453.845,A -85,B 0,C 180,E1 -5633.005,E2 -5633.005} C_VEL
LIN {X 0,Y 502.767,Z 453.855,A -85,B 0,C 180,E1 -5633.231,E2 -5633.231} C_VEL
LIN {X 0,Y 502.81,Z 453.856,A -85,B 0,C 180,E1 -5636.006,E2 -5636.006} C_VEL
LIN {X 0,Y 502.801,Z 453.854,A -85,B 0,C 180,E1 -5638.857,E2 -5638.857} C_VEL
LIN {X 0,Y 502.849,Z 453.847,A -85,B 0,C 180,E1 -5641.705,E2 -5641.705} C_VEL
LIN {X 0,Y 502.827,Z 453.854,A -85,B 0,C 180,E1 -5644.324,E2 -5644.324} C_VEL
LIN {X 0,Y 502.809,Z 453.851,A -85,B 0,C 180,E1 -5647.298,E2 -5647.298} C_VEL
LIN {X 0,Y 502.83,Z 453.849,A -85,B 0,C 180,E1 -5650.4,E2 -5650.4} C_VEL
LIN {X 0,Y 502.825,Z 453.853,A -85,B 0,C 180,E1 -5652.931,E2 -5652.931} C_VEL
LIN {X 0,Y 502.851,Z 453.846,A -85,B 0,C 180,E1 -5655.429,E2 -5655.429} C_VEL
LIN {X 0,Y 502.883,Z 453.841,A -85,B 0,C 180,E1 -5658.717,E2 -5658.717} C_VEL
LIN {X 0,Y 502.907,Z 453.841,A -85,B 0,C 180,E1 -5661.967,E2 -5661.967} C_VEL
LIN {X 0,Y 502.942,Z 453.836,A -85,B 0,C 180,E1 -5664.387,E2 -5664.387} C_VEL
LIN {X 0,Y 503.03,Z 453.824,A -85,B 0,C 180,E1 -5667.598,E2 -5667.598} C_VEL
LIN {X 0,Y 503.034,Z 453.827,A -85,B 0,C 180,E1 -5670,E2 -5670} C_VEL
LIN {X 0,Y 503.03,Z 453.824,A -85,B 0,C 180,E1 -5672.402,E2 -5672.402} C_VEL
LIN {X 0,Y 502.933,Z 453.839,A -85,B 0,C 180,E1 -5675.614,E2 -5675.614} C_VEL
LIN {X 0,Y 502.87,Z 453.847,A -85,B 0,C 180,E1 -5678.843,E2 -5678.843} C_VEL
LIN {X 0,Y 502.852,Z 453.851,A -85,B 0,C 180,E1 -5682.102,E2 -5682.102} C_VEL
LIN {X 0,Y 502.855,Z 453.848,A -85,B 0,C 180,E1 -5685.4,E2 -5685.4} C_VEL
LIN {X 0,Y 502.847,Z 453.847,A -85,B 0,C 180,E1 -5688.12,E2 -5688.12} C_VEL
LIN {X 0,Y 502.835,Z 453.852,A -85,B 0,C 180,E1 -5690.536,E2 -5690.536} C_VEL
LIN {X 0,Y 502.794,Z 453.854,A -85,B 0,C 180,E1 -5693.041,E2 -5693.041} C_VEL
LIN {X 0,Y 502.827,Z 453.852,A -85,B 0,C 180,E1 -5695.676,E2 -5695.676} C_VEL
LIN {X 0,Y 502.845,Z 453.846,A -85,B 0,C 180,E1 -5698.373,E2 -5698.373} C_VEL
LIN {X 0,Y 502.798,Z 453.855,A -85,B 0,C 180,E1 -5701.499,E2 -5701.499} C_VEL
LIN {X 0,Y 502.81,Z 453.855,A -85,B 0,C 180,E1 -5704.444,E2 -5704.444} C_VEL
LIN {X 0,Y 502.785,Z 453.854,A -85,B 0,C 180,E1 -5707.178,E2 -5707.178} C_VEL
LIN {X 0,Y 502.792,Z 453.855,A -85,B 0,C 180,E1 -5710.015,E2 -5710.015} C_VEL
LIN {X 0,Y 502.807,Z 453.851,A -85,B 0,C 180,E1 -5712.199,E2 -5712.199} C_VEL
LIN {X 0,Y 502.806,Z 453.853,A -85,B 0,C 180,E1 -5715.468,E2 -5715.468} C_VEL
LIN {X 0,Y 502.835,Z 453.85,A -85,B 0,C 180,E1 -5717.864,E2 -5717.864} C_VEL
LIN {X 0,Y 502.805,Z 453.851,A -85,B 0,C 180,E1 -5721.024,E2 -5721.024} C_VEL
LIN {X 0,Y 502.757,Z 453.858,A -85,B 0,C 180,E1 -5724.172,E2 -5724.172} C_VEL
LIN {X 0,Y 502.557,Z 453.887,A -85,B 0,C 180,E1 -5727.042,E2 -5727.042} C_VEL
LIN {X 0,Y 502.337,Z 453.915,A -85,B 0,C 180,E1 -5728.825,E2 -5728.825} C_VEL
LIN {X 0,Y 502.224,Z 454.961,A -85,B 0,C 180,E1 -5730.183,E2 -5730.183} C_VEL
LIN {X 0,Y 502.272,Z 458.726,A -85,B 0,C 180,E1 -5733.4,E2 -5733.4} C_VEL
LIN {X 0,Y 502.202,Z 461.827,A -85,B 0,C 180,E1 -5736.056,E2 -5736.056} C_VEL
LIN {X 0,Y 502.162,Z 464.811,A -85,B 0,C 180,E1 -5738.661,E2 -5738.661} C_VEL
LIN {X 0,Y 502.124,Z 467.76,A -85,B 0,C 180,E1 -5741.221,E2 -5741.221} C_VEL
LIN {X 0,Y 502.108,Z 470.683,A -85,B 0,C 180,E1 -5743.743,E2 -5743.743} C_VEL
LIN {X 0,Y 502.161,Z 473.097,A -85,B 0,C 180,E1 -5745.835,E2 -5745.835} C_VEL
LIN {X 0,Y 504.503,Z 485.498,A -85,B 0,C 180,E1 -5746.249,E2 -5746.249} C_VEL
LIN {X 0,Y 504.337,Z 498.002,A -85,B 0,C 180,E1 -5746.758,E2 -5746.758} C_VEL
LIN {X 0,Y 504.031,Z 510.451,A -85,B 0,C 180,E1 -5747.437,E2 -5747.437} C_VEL
LIN {X 0,Y 503.703,Z 521.635,A -85,B 0,C 180,E1 -5748.225,E2 -5748.225} C_VEL
LIN {X 0,Y 503.272,Z 532.981,A -85,B 0,C 180,E1 -5749.235,E2 -5749.235} C_VEL
LIN {X 0,Y 503.013,Z 541.285,A -85,B 0,C 180,E1 -5750.145,E2 -5750.145} C_VEL
LIN {X 0,Y 502.772,Z 548.96,A -85,B 0,C 180,E1 -5751.155,E2 -5751.155} C_VEL
LIN {X 0,Y 502.494,Z 556.443,A -85,B 0,C 180,E1 -5752.364,E2 -5752.364} C_VEL
LIN {X 0,Y 502.324,Z 562.444,A -85,B 0,C 180,E1 -5753.573,E2 -5753.573} C_VEL
LIN {X 0,Y 502.188,Z 567.194,A -85,B 0,C 180,E1 -5754.781,E2 -5754.781} C_VEL
LIN {X 0,Y 502.237,Z 570.826,A -85,B 0,C 180,E1 -5755.988,E2 -5755.988} C_VEL
LIN {X 0,Y 502.125,Z 572.704,A -85,B 0,C 180,E1 -5756.79,E2 -5756.79} C_VEL
LIN {X 0,Y 502.12,Z 574.142,A -85,B 0,C 180,E1 -5757.593,E2 -5757.593} C_VEL
LIN {X 0,Y 501.991,Z 575.783,A -85,B 0,C 180,E1 -5759.198,E2 -5759.198} C_VEL
LIN {X 0,Y 501.983,Z 576.033,A -85,B 0,C 180,E1 -5760,E2 -5760} C_VEL
LIN {X 0,Y 501.991,Z 575.854,A -85,B 0,C 180,E1 -5760.802,E2 -5760.802} C_VEL
LIN {X 0,Y 502.121,Z 574.32,A -85,B 0,C 180,E1 -5762.406,E2 -5762.406} C_VEL
LIN {X 0,Y 502.137,Z 572.968,A -85,B 0,C 180,E1 -5763.209,E2 -5763.209} C_VEL
LIN {X 0,Y 502.21,Z 570.114,A -85,B 0,C 180,E1 -5764.414,E2 -5764.414} C_VEL
LIN {X 0,Y 502.283,Z 566.229,A -85,B 0,C 180,E1 -5765.621,E2 -5765.621} C_VEL
LIN {X 0,Y 502.401,Z 560.647,A -85,B 0,C 180,E1 -5766.94,E2 -5766.94} C_VEL
LIN {X 0,Y 502.613,Z 553.626,A -85,B 0,C 180,E1 -5768.24,E2 -5768.24} C_VEL
LIN {X 0,Y 502.842,Z 545.422,A -85,B 0,C 180,E1 -5769.452,E2 -5769.452} C_VEL
LIN {X 0,Y 503.132,Z 536.968,A -85,B 0,C 180,E1 -5770.462,E2 -5770.462} C_VEL
LIN {X 0,Y 503.55,Z 526.588,A -85,B 0,C 180,E1 -5771.472,E2 -5771.472} C_VEL
LIN {X 0,Y 503.902,Z 516.074,A -85,B 0,C 180,E1 -5772.295,E2 -5772.295} C_VEL
LIN {X 0,Y 504.186,Z 504.882,A -85,B 0,C 180,E1 -5772.989,E2 -5772.989} C_VEL
LIN {X 0,Y 504.505,Z 492.118,A -85,B 0,C 180,E1 -5773.596,E2 -5773.596} C_VEL
LIN {X 0,Y 504.377,Z 484.776,A -85,B 0,C 180,E1 -5773.869,E2 -5773.869} C_VEL
LIN {X 0,Y 502.218,Z 473.808,A -85,B 0,C 180,E1 -5774.253,E2 -5774.253} C_VEL
LIN {X 0,Y 502.207,Z 470.57,A -85,B 0,C 180,E1 -5777.09,E2 -5777.09} C_VEL
LIN {X 0,Y 502.241,Z 466.758,A -85,B 0,C 180,E1 -5780.355,E2 -5780.355} C_VEL
LIN {X 0,Y 502.196,Z 463.611,A -85,B 0,C 180,E1 -5783.069,E2 -5783.069} C_VEL
LIN {X 0,Y 502.255,Z 460.316,A -85,B 0,C 180,E1 -5785.708,E2 -5785.708} C_VEL
LIN {X 0,Y 502.206,Z 456.647,A -85,B 0,C 180,E1 -5788.412,E2 -5788.412} C_VEL
LIN {X 0,Y 502.2,Z 454.06,A -85,B 0,C 180,E1 -5790.252,E2 -5790.252} C_VEL
LIN {X 0,Y 502.57,Z 453.887,A -85,B 0,C 180,E1 -5793.051,E2 -5793.051} C_VEL
LIN {X 0,Y 502.759,Z 453.862,A -85,B 0,C 180,E1 -5795.952,E2 -5795.952} C_VEL
LIN {X 0,Y 502.803,Z 453.854,A -85,B 0,C 180,E1 -5798.976,E2 -5798.976} C_VEL
LIN {X 0,Y 502.833,Z 453.853,A -85,B 0,C 180,E1 -5802.136,E2 -5802.136} C_VEL
LIN {X 0,Y 502.803,Z 453.855,A -85,B 0,C 180,E1 -5805.468,E2 -5805.468} C_VEL
LIN {X 0,Y 502.822,Z 453.853,A -85,B 0,C 180,E1 -5808.934,E2 -5808.934} C_VEL
LIN {X 0,Y 502.836,Z 453.988,A -85,B 0,C 180,E1 -5810.769,E2 -5810.769} C_VEL
LIN {X 0,Y 504.031,Z 460.921,A -85,B 0,C 180,E1 -5813.598,E2 -5813.598} C_VEL
LIN {X 0,Y 504.187,Z 465.434,A -85,B 0,C 180,E1 -5815.328,E2 -5815.328} C_VEL
LIN {X 0,Y 503.835,Z 473.578,A -85,B 0,C 180,E1 -5818.309,E2 -5818.309} C_VEL
LIN {X 0,Y 503.456,Z 481.796,A -85,B 0,C 180,E1 -5821.21,E2 -5821.21} C_VEL
LIN {X 0,Y 503.218,Z 489.643,A -85,B 0,C 180,E1 -5823.9,E2 -5823.9} C_VEL
LIN {X 0,Y 502.908,Z 498.856,A -85,B 0,C 180,E1 -5826.965,E2 -5826.965} C_VEL
LIN {X 0,Y 502.716,Z 508.129,A -85,B 0,C 180,E1 -5829.97,E2 -5829.97} C_VEL
LIN {X 0,Y 502.548,Z 517.452,A -85,B 0,C 180,E1 -5832.922,E2 -5832.922} C_VEL
LIN {X 0,Y 502.403,Z 526.386,A -85,B 0,C 180,E1 -5835.701,E2 -5835.701} C_VEL
LIN {X 0,Y 504.558,Z 540.738,A -85,B 0,C 180,E1 -5836.123,E2 -5836.123} C_VEL
LIN {X 0,Y 504.31,Z 553.388,A -85,B 0,C 180,E1 -5836.604,E2 -5836.604} C_VEL
LIN {X 0,Y 503.965,Z 566.21,A -85,B 0,C 180,E1 -5837.27,E2 -5837.27} C_VEL
LIN {X 0,Y 503.581,Z 577.329,A -85,B 0,C 180,E1 -5838.018,E2 -5838.018} C_VEL
LIN {X 0,Y 503.238,Z 588.101,A -85,B 0,C 180,E1 -5838.929,E2 -5838.929} C_VEL
LIN {X 0,Y 502.888,Z 597.809,A -85,B 0,C 180,E1 -5839.939,E2 -5839.939} C_VEL
LIN {X 0,Y 502.661,Z 605.781,A -85,B 0,C 180,E1 -5840.95,E2 -5840.95} C_VEL
LIN {X 0,Y 502.416,Z 613.575,A -85,B 0,C 180,E1 -5842.161,E2 -5842.161} C_VEL
LIN {X 0,Y 502.228,Z 620.367,A -85,B 0,C 180,E1 -5843.49,E2 -5843.49} C_VEL
LIN {X 0,Y 502.183,Z 625.516,A -85,B 0,C 180,E1 -5844.781,E2 -5844.781} C_VEL
LIN {X 0,Y 502.165,Z 629.164,A -85,B 0,C 180,E1 -5845.987,E2 -5845.987} C_VEL
LIN {X 0,Y 502.121,Z 631.042,A -85,B 0,C 180,E1 -5846.791,E2 -5846.791} C_VEL
LIN {X 0,Y 502.12,Z 632.452,A -85,B 0,C 180,E1 -5847.593,E2 -5847.593} C_VEL
LIN {X 0,Y 501.99,Z 634.059,A -85,B 0,C 180,E1 -5849.198,E2 -5849.198} C_VEL
LIN {X 0,Y 501.98,Z 634.27,A -85,B 0,C 180,E1 -5850,E2 -5850} C_VEL
LIN {X 0,Y 502.036,Z 633.431,A -85,B 0,C 180,E1 -5851.604,E2 -5851.604} C_VEL
LIN {X 0,Y 502.12,Z 632.423,A -85,B 0,C 180,E1 -5852.407,E2 -5852.407} C_VEL
LIN {X 0,Y 502.121,Z 630.994,A -85,B 0,C 180,E1 -5853.209,E2 -5853.209} C_VEL
LIN {X 0,Y 502.127,Z 628.006,A -85,B 0,C 180,E1 -5854.415,E2 -5854.415} C_VEL
LIN {X 0,Y 502.238,Z 623.966,A -85,B 0,C 180,E1 -5855.621,E2 -5855.621} C_VEL
LIN {X 0,Y 502.332,Z 617.845,A -85,B 0,C 180,E1 -5857.012,E2 -5857.012} C_VEL
LIN {X 0,Y 502.499,Z 610.947,A -85,B 0,C 180,E1 -5858.242,E2 -5858.242} C_VEL
LIN {X 0,Y 502.728,Z 602.501,A -85,B 0,C 180,E1 -5859.454,E2 -5859.454} C_VEL
LIN {X 0,Y 503.013,Z 593.83,A -85,B 0,C 180,E1 -5860.465,E2 -5860.465} C_VEL
LIN {X 0,Y 503.342,Z 583.141,A -85,B 0,C 180,E1 -5861.477,E2 -5861.477} C_VEL
LIN {X 0,Y 503.672,Z 572.164,A -85,B 0,C 180,E1 -5862.315,E2 -5862.315} C_VEL
LIN {X 0,Y 504.034,Z 559.973,A -85,B 0,C 180,E1 -5863.045,E2 -5863.045} C_VEL
LIN {X 0,Y 504.379,Z 546.463,A -85,B 0,C 180,E1 -5863.651,E2 -5863.651} C_VEL
LIN {X 0,Y 504.29,Z 539.438,A -85,B 0,C 180,E1 -5863.898,E2 -5863.898} C_VEL
LIN {X 0,Y 502.452,Z 526.623,A -85,B 0,C 180,E1 -5864.262,E2 -5864.262} C_VEL
LIN {X 0,Y 502.406,Z 525.612,A -85,B 0,C 180,E1 -5864.325,E2 -5864.325} C_VEL
LIN {X 0,Y 502.476,Z 516.496,A -85,B 0,C 180,E1 -5867.081,E2 -5867.081} C_VEL
LIN {X 0,Y 502.691,Z 505.495,A -85,B 0,C 180,E1 -5870.458,E2 -5870.458} C_VEL
LIN {X 0,Y 502.831,Z 495.97,A -85,B 0,C 180,E1 -5873.475,E2 -5873.475} C_VEL
LIN {X 0,Y 503.052,Z 486.532,A -85,B 0,C 180,E1 -5876.603,E2 -5876.603} C_VEL
LIN {X 0,Y 503.272,Z 478.986,A -85,B 0,C 180,E1 -5879.259,E2 -5879.259} C_VEL
LIN {X 0,Y 503.621,Z 472.644,A -85,B 0,C 180,E1 -5881.652,E2 -5881.652} C_VEL
LIN {X 0,Y 503.988,Z 467.187,A -85,B 0,C 180,E1 -5883.903,E2 -5883.903} C_VEL
LIN {X 0,Y 504.199,Z 462.566,A -85,B 0,C 180,E1 -5886.054,E2 -5886.054} C_VEL
LIN {X 0,Y 503.793,Z 459.338,A -85,B 0,C 180,E1 -5887.866,E2 -5887.866} C_VEL
LIN {X 0,Y 503.238,Z 456.303,A -85,B 0,C 180,E1 -5889.972,E2 -5889.972} C_VEL
LIN {X 0,Y 502.832,Z 453.952,A -85,B 0,C 180,E1 -5892.203,E2 -5892.203} C_VEL
LIN {X 0,Y 502.803,Z 453.857,A -85,B 0,C 180,E1 -5895.468,E2 -5895.468} C_VEL
LIN {X 0,Y 502.833,Z 453.853,A -85,B 0,C 180,E1 -5897.864,E2 -5897.864} C_VEL
LIN {X 0,Y 502.805,Z 453.857,A -85,B 0,C 180,E1 -5901.024,E2 -5901.024} C_VEL
LIN {X 0,Y 502.755,Z 453.877,A -85,B 0,C 180,E1 -5903.052,E2 -5903.052} C_VEL
LIN {X 0,Y 502.856,Z 455.487,A -85,B 0,C 180,E1 -5905.548,E2 -5905.548} C_VEL
LIN {X 0,Y 502.729,Z 457.755,A -85,B 0,C 180,E1 -5908.514,E2 -5908.514} C_VEL
LIN {X 0,Y 502.589,Z 460.472,A -85,B 0,C 180,E1 -5911.76,E2 -5911.76} C_VEL
LIN {X 0,Y 502.482,Z 462.752,A -85,B 0,C 180,E1 -5914.305,E2 -5914.305} C_VEL
LIN {X 0,Y 502.371,Z 465.645,A -85,B 0,C 180,E1 -5917.417,E2 -5917.417} C_VEL
LIN {X 0,Y 502.274,Z 468.517,A -85,B 0,C 180,E1 -5920.378,E2 -5920.378} C_VEL
LIN {X 0,Y 502.241,Z 471.053,A -85,B 0,C 180,E1 -5922.911,E2 -5922.911} C_VEL
LIN {X 0,Y 502.223,Z 474.102,A -85,B 0,C 180,E1 -5925.85,E2 -5925.85} C_VEL
LIN {X 0,Y 504.358,Z 484.724,A -85,B 0,C 180,E1 -5926.207,E2 -5926.207} C_VEL
LIN {X 0,Y 504.578,Z 488.757,A -85,B 0,C 180,E1 -5926.355,E2 -5926.355} C_VEL
LIN {X 0,Y 504.296,Z 501.481,A -85,B 0,C 180,E1 -5926.911,E2 -5926.911} C_VEL
LIN {X 0,Y 503.997,Z 513.634,A -85,B 0,C 180,E1 -5927.621,E2 -5927.621} C_VEL
LIN {X 0,Y 503.635,Z 524.495,A -85,B 0,C 180,E1 -5928.428,E2 -5928.428} C_VEL
LIN {X 0,Y 503.292,Z 534.306,A -85,B 0,C 180,E1 -5929.338,E2 -5929.338} C_VEL
LIN {X 0,Y 502.99,Z 543.217,A -85,B 0,C 180,E1 -5930.348,E2 -5930.348} C_VEL
LIN {X 0,Y 502.703,Z 551.907,A -85,B 0,C 180,E1 -5931.559,E2 -5931.559} C_VEL
LIN {X 0,Y 502.468,Z 558.831,A -85,B 0,C 180,E1 -5932.768,E2 -5932.768} C_VEL
LIN {X 0,Y 502.362,Z 564.351,A -85,B 0,C 180,E1 -5933.977,E2 -5933.977} C_VEL
LIN {X 0,Y 502.138,Z 568.69,A -85,B 0,C 180,E1 -5935.183,E2 -5935.183} C_VEL
LIN {X 0,Y 502.236,Z 570.967,A -85,B 0,C 180,E1 -5935.988,E2 -5935.988} C_VEL
LIN {X 0,Y 502.137,Z 572.831,A -85,B 0,C 180,E1 -5936.791,E2 -5936.791} C_VEL
LIN {X 0,Y 502.121,Z 574.237,A -85,B 0,C 180,E1 -5937.594,E2 -5937.594} C_VEL
LIN {X 0,Y 501.991,Z 575.843,A -85,B 0,C 180,E1 -5939.198,E2 -5939.198} C_VEL
LIN {X 0,Y 501.982,Z 576.07,A -85,B 0,C 180,E1 -5940,E2 -5940} C_VEL
LIN {X 0,Y 501.991,Z 575.877,A -85,B 0,C 180,E1 -5940.802,E2 -5940.802} C_VEL
LIN {X 0,Y 502.12,Z 574.302,A -85,B 0,C 180,E1 -5942.407,E2 -5942.407} C_VEL
LIN {X 0,Y 502.125,Z 572.933,A -85,B 0,C 180,E1 -5943.21,E2 -5943.21} C_VEL
LIN {X 0,Y 502.209,Z 570.045,A -85,B 0,C 180,E1 -5944.415,E2 -5944.415} C_VEL
LIN {X 0,Y 502.282,Z 566.134,A -85,B 0,C 180,E1 -5945.621,E2 -5945.621} C_VEL
LIN {X 0,Y 502.39,Z 561.088,A -85,B 0,C 180,E1 -5946.829,E2 -5946.829} C_VEL
LIN {X 0,Y 502.554,Z 554.721,A -85,B 0,C 180,E1 -5948.039,E2 -5948.039} C_VEL
LIN {X 0,Y 502.768,Z 546.766,A -85,B 0,C 180,E1 -5949.251,E2 -5949.251} C_VEL
LIN {X 0,Y 503.095,Z 538.642,A -85,B 0,C 180,E1 -5950.26,E2 -5950.26} C_VEL
LIN {X 0,Y 503.451,Z 528.735,A -85,B 0,C 180,E1 -5951.27,E2 -5951.27} C_VEL
LIN {X 0,Y 503.818,Z 517.607,A -85,B 0,C 180,E1 -5952.176,E2 -5952.176} C_VEL
LIN {X 0,Y 504.092,Z 506.616,A -85,B 0,C 180,E1 -5952.89,E2 -5952.89} C_VEL
LIN {X 0,Y 504.425,Z 494.57,A -85,B 0,C 180,E1 -5953.496,E2 -5953.496} C_VEL
LIN {X 0,Y 504.476,Z 485.614,A -85,B 0,C 180,E1 -5953.841,E2 -5953.841} C_VEL
LIN {X 0,Y 502.462,Z 474.698,A -85,B 0,C 180,E1 -5954.213,E2 -5954.213} C_VEL
LIN {X 0,Y 502.172,Z 473.165,A -85,B 0,C 180,E1 -5954.281,E2 -5954.281} C_VEL
LIN {X 0,Y 502.182,Z 469.049,A -85,B 0,C 180,E1 -5957.932,E2 -5957.932} C_VEL
LIN {X 0,Y 502.176,Z 466.214,A -85,B 0,C 180,E1 -5960.48,E2 -5960.48} C_VEL
LIN {X 0,Y 502.194,Z 463.363,A -85,B 0,C 180,E1 -5963.07,E2 -5963.07} C_VEL
LIN {X 0,Y 502.271,Z 460.465,A -85,B 0,C 180,E1 -5965.707,E2 -5965.707} C_VEL
LIN {X 0,Y 502.303,Z 457.531,A -85,B 0,C 180,E1 -5968.406,E2 -5968.406} C_VEL
LIN {X 0,Y 502.333,Z 454.304,A -85,B 0,C 180,E1 -5971.412,E2 -5971.412} C_VEL
LIN {X 0,Y 502.376,Z 453.911,A -85,B 0,C 180,E1 -5972.114,E2 -5972.114} C_VEL
LIN {X 0,Y 502.686,Z 453.871,A -85,B 0,C 180,E1 -5974.975,E2 -5974.975} C_VEL
LIN {X 0,Y 502.795,Z 453.853,A -85,B 0,C 180,E1 -5977.954,E2 -5977.954} C_VEL
LIN {X 0,Y 502.825,Z 453.848,A -85,B 0,C 180,E1 -5981.066,E2 -5981.066} C_VEL
LIN {X 0,Y 502.787,Z 453.855,A -85,B 0,C 180,E1 -5983.376,E2 -5983.376} C_VEL
LIN {X 0,Y 502.795,Z 453.857,A -85,B 0,C 180,E1 -5985.661,E2 -5985.661} C_VEL
LIN {X 0,Y 502.823,Z 453.853,A -85,B 0,C 180,E1 -5989.005,E2 -5989.005} C_VEL
LIN {X 0,Y 502.798,Z 453.854,A -85,B 0,C 180,E1 -5992.046,E2 -5992.046} C_VEL
LIN {X 0,Y 502.767,Z 453.855,A -85,B 0,C 180,E1 -5993.231,E2 -5993.231} C_VEL
LIN {X 0,Y 502.101,Z 453.943,A -85,B 0,C 180,E1 -5993.9,E2 -5993.9} C_VEL
LIN {X 0,Y 499.306,Z 454.288,A -85,B 0,C 180,E1 -5994.987,E2 -5994.987} C_VEL
LIN {X 0,Y 496.934,Z 454.588,A -85,B 0,C 180,E1 -5995.863,E2 -5995.863} C_VEL
LIN {X 0,Y 495.894,Z 454.714,A -85,B 0,C 180,E1 -5996.539,E2 -5996.539} C_VEL
LIN {X 0,Y 495.797,Z 454.725,A -85,B 0,C 180,E1 -5996.768,E2 -5996.768} C_VEL
LIN {X 0,Y 495.77,Z 454.729,A -85,B 0,C 180,E1 -5999.853,E2 -5999.853} C_VEL
LIN {X 0,Y 495.819,Z 454.724,A -85,B 0,C 180,E1 -6003.026,E2 -6003.026} C_VEL
LIN {X 0,Y 495.738,Z 454.733,A -85,B 0,C 180,E1 -6005.724,E2 -6005.724} C_VEL
LIN {X 0,Y 495.748,Z 454.732,A -85,B 0,C 180,E1 -6008.371,E2 -6008.371} C_VEL
LIN {X 0,Y 495.788,Z 454.729,A -85,B 0,C 180,E1 -6010.972,E2 -6010.972} C_VEL
LIN {X 0,Y 495.813,Z 454.726,A -85,B 0,C 180,E1 -6014.376,E2 -6014.376} C_VEL
LIN {X 0,Y 495.789,Z 454.727,A -85,B 0,C 180,E1 -6016.891,E2 -6016.891} C_VEL
LIN {X 0,Y 495.779,Z 454.727,A -85,B 0,C 180,E1 -6019.381,E2 -6019.381} C_VEL
LIN {X 0,Y 495.878,Z 454.718,A -85,B 0,C 180,E1 -6021.852,E2 -6021.852} C_VEL
LIN {X 0,Y 495.9,Z 454.713,A -85,B 0,C 180,E1 -6024.307,E2 -6024.307} C_VEL
LIN {X 0,Y 495.999,Z 454.7,A -85,B 0,C 180,E1 -6027.564,E2 -6027.564} C_VEL
LIN {X 0,Y 495.989,Z 454.7,A -85,B 0,C 180,E1 -6030.812,E2 -6030.812} C_VEL
LIN {X 0,Y 495.999,Z 454.7,A -85,B 0,C 180,E1 -6032.436,E2 -6032.436} C_VEL
LIN {X 0,Y 495.888,Z 454.716,A -85,B 0,C 180,E1 -6035.694,E2 -6035.694} C_VEL
LIN {X 0,Y 495.84,Z 454.722,A -85,B 0,C 180,E1 -6038.97,E2 -6038.97} C_VEL
LIN {X 0,Y 495.835,Z 454.724,A -85,B 0,C 180,E1 -6042.035,E2 -6042.035} C_VEL
LIN {X 0,Y 495.83,Z 454.723,A -85,B 0,C 180,E1 -6045.452,E2 -6045.452} C_VEL
LIN {X 0,Y 495.813,Z 454.723,A -85,B 0,C 180,E1 -6048.247,E2 -6048.247} C_VEL
LIN {X 0,Y 495.78,Z 454.73,A -85,B 0,C 180,E1 -6050.756,E2 -6050.756} C_VEL
LIN {X 0,Y 495.748,Z 454.731,A -85,B 0,C 180,E1 -6053.387,E2 -6053.387} C_VEL
LIN {X 0,Y 495.829,Z 454.719,A -85,B 0,C 180,E1 -6056.749,E2 -6056.749} C_VEL
LIN {X 0,Y 495.772,Z 454.73,A -85,B 0,C 180,E1 -6059.746,E2 -6059.746} C_VEL
LIN {X 0,Y 495.773,Z 454.731,A -85,B 0,C 180,E1 -6062.594,E2 -6062.594} C_VEL
LIN {X 0,Y 495.76,Z 454.73,A -85,B 0,C 180,E1 -6065.537,E2 -6065.537} C_VEL
LIN {X 0,Y 495.768,Z 454.727,A -85,B 0,C 180,E1 -6068.768,E2 -6068.768} C_VEL
LIN {X 0,Y 495.761,Z 454.731,A -85,B 0,C 180,E1 -6071.781,E2 -6071.781} C_VEL
LIN {X 0,Y 495.754,Z 454.733,A -85,B 0,C 180,E1 -6075.139,E2 -6075.139} C_VEL
LIN {X 0,Y 495.782,Z 454.731,A -85,B 0,C 180,E1 -6078.221,E2 -6078.221} C_VEL
LIN {X 0,Y 495.754,Z 454.732,A -85,B 0,C 180,E1 -6081.408,E2 -6081.408} C_VEL
LIN {X 0,Y 495.687,Z 454.739,A -85,B 0,C 180,E1 -6084.457,E2 -6084.457} C_VEL
LIN {X 0,Y 495.47,Z 454.771,A -85,B 0,C 180,E1 -6087.383,E2 -6087.383} C_VEL
LIN {X 0,Y 495.22,Z 454.802,A -85,B 0,C 180,E1 -6089.276,E2 -6089.276} C_VEL
LIN {X 0,Y 495.139,Z 456.685,A -85,B 0,C 180,E1 -6091.144,E2 -6091.144} C_VEL
LIN {X 0,Y 495.19,Z 459.88,A -85,B 0,C 180,E1 -6093.898,E2 -6093.898} C_VEL
LIN {X 0,Y 495.093,Z 462.992,A -85,B 0,C 180,E1 -6096.58,E2 -6096.58} C_VEL
LIN {X 0,Y 495.115,Z 466.386,A -85,B 0,C 180,E1 -6099.53,E2 -6099.53} C_VEL
LIN {X 0,Y 495.067,Z 469.951,A -85,B 0,C 180,E1 -6102.655,E2 -6102.655} C_VEL
LIN {X 0,Y 495.058,Z 473.41,A -85,B 0,C 180,E1 -6105.634,E2 -6105.634} C_VEL
LIN {X 0,Y 497.475,Z 485.572,A -85,B 0,C 180,E1 -6106.051,E2 -6106.051} C_VEL
LIN {X 0,Y 497.526,Z 495.951,A -85,B 0,C 180,E1 -6106.469,E2 -6106.469} C_VEL
LIN {X 0,Y 497.164,Z 507.978,A -85,B 0,C 180,E1 -6107.097,E2 -6107.097} C_VEL
LIN {X 0,Y 496.773,Z 520.538,A -85,B 0,C 180,E1 -6107.955,E2 -6107.955} C_VEL
LIN {X 0,Y 496.386,Z 531.134,A -85,B 0,C 180,E1 -6108.877,E2 -6108.877} C_VEL
LIN {X 0,Y 496.003,Z 541.537,A -85,B 0,C 180,E1 -6110.004,E2 -6110.004} C_VEL
LIN {X 0,Y 495.744,Z 549.238,A -85,B 0,C 180,E1 -6111.028,E2 -6111.028} C_VEL
LIN {X 0,Y 495.469,Z 556.749,A -85,B 0,C 180,E1 -6112.255,E2 -6112.255} C_VEL
LIN {X 0,Y 495.273,Z 562.77,A -85,B 0,C 180,E1 -6113.481,E2 -6113.481} C_VEL
LIN {X 0,Y 495.129,Z 567.54,A -85,B 0,C 180,E1 -6114.706,E2 -6114.706} C_VEL
LIN {X 0,Y 495.171,Z 571.188,A -85,B 0,C 180,E1 -6115.93,E2 -6115.93} C_VEL
LIN {X 0,Y 495.051,Z 573.078,A -85,B 0,C 180,E1 -6116.744,E2 -6116.744} C_VEL
LIN {X 0,Y 495.054,Z 574.523,A -85,B 0,C 180,E1 -6117.559,E2 -6117.559} C_VEL
LIN {X 0,Y 494.911,Z 576.177,A -85,B 0,C 180,E1 -6119.186,E2 -6119.186} C_VEL
LIN {X 0,Y 494.901,Z 576.431,A -85,B 0,C 180,E1 -6120,E2 -6120} C_VEL
LIN {X 0,Y 494.911,Z 576.254,A -85,B 0,C 180,E1 -6120.813,E2 -6120.813} C_VEL
LIN {X 0,Y 495.055,Z 574.721,A -85,B 0,C 180,E1 -6122.441,E2 -6122.441} C_VEL
LIN {X 0,Y 495.062,Z 573.366,A -85,B 0,C 180,E1 -6123.255,E2 -6123.255} C_VEL
LIN {X 0,Y 495.14,Z 570.505,A -85,B 0,C 180,E1 -6124.477,E2 -6124.477} C_VEL
LIN {X 0,Y 495.228,Z 566.61,A -85,B 0,C 180,E1 -6125.701,E2 -6125.701} C_VEL
LIN {X 0,Y 495.37,Z 560.668,A -85,B 0,C 180,E1 -6127.11,E2 -6127.11} C_VEL
LIN {X 0,Y 495.605,Z 553.97,A -85,B 0,C 180,E1 -6128.358,E2 -6128.358} C_VEL
LIN {X 0,Y 495.849,Z 545.733,A -85,B 0,C 180,E1 -6129.587,E2 -6129.587} C_VEL
LIN {X 0,Y 496.149,Z 537.253,A -85,B 0,C 180,E1 -6130.611,E2 -6130.611} C_VEL
LIN {X 0,Y 496.61,Z 526.842,A -85,B 0,C 180,E1 -6131.634,E2 -6131.634} C_VEL
LIN {X 0,Y 496.964,Z 515.414,A -85,B 0,C 180,E1 -6132.528,E2 -6132.528} C_VEL
LIN {X 0,Y 497.325,Z 503.186,A -85,B 0,C 180,E1 -6133.276,E2 -6133.276} C_VEL
LIN {X 0,Y 497.646,Z 490.906,A -85,B 0,C 180,E1 -6133.839,E2 -6133.839} C_VEL
LIN {X 0,Y 497.388,Z 485.221,A -85,B 0,C 180,E1 -6134.055,E2 -6134.055} C_VEL
LIN {X 0,Y 495.156,Z 474.289,A -85,B 0,C 180,E1 -6134.434,E2 -6134.434} C_VEL
LIN {X 0,Y 495.173,Z 470.169,A -85,B 0,C 180,E1 -6138.022,E2 -6138.022} C_VEL
LIN {X 0,Y 495.155,Z 466.94,A -85,B 0,C 180,E1 -6140.783,E2 -6140.783} C_VEL
LIN {X 0,Y 495.147,Z 463.789,A -85,B 0,C 180,E1 -6143.417,E2 -6143.417} C_VEL
LIN {X 0,Y 495.206,Z 460.407,A -85,B 0,C 180,E1 -6146.101,E2 -6146.101} C_VEL
LIN {X 0,Y 495.12,Z 456.737,A -85,B 0,C 180,E1 -6148.856,E2 -6148.856} C_VEL
LIN {X 0,Y 495.155,Z 455.107,A -85,B 0,C 180,E1 -6150.025,E2 -6150.025} C_VEL
LIN {X 0,Y 495.366,Z 454.784,A -85,B 0,C 180,E1 -6151.664,E2 -6151.664} C_VEL
LIN {X 0,Y 495.676,Z 454.744,A -85,B 0,C 180,E1 -6154.678,E2 -6154.678} C_VEL
LIN {X 0,Y 495.731,Z 454.735,A -85,B 0,C 180,E1 -6157.562,E2 -6157.562} C_VEL
LIN {X 0,Y 495.769,Z 454.732,A -85,B 0,C 180,E1 -6160.7,E2 -6160.7} C_VEL
LIN {X 0,Y 495.738,Z 454.736,A -85,B 0,C 180,E1 -6163.695,E2 -6163.695} C_VEL
LIN {X 0,Y 495.731,Z 454.736,A -85,B 0,C 180,E1 -6166.305,E2 -6166.305} C_VEL
LIN {X 0,Y 495.769,Z 454.732,A -85,B 0,C 180,E1 -6169.3,E2 -6169.3} C_VEL
LIN {X 0,Y 495.783,Z 454.785,A -85,B 0,C 180,E1 -6170.476,E2 -6170.476} C_VEL
LIN {X 0,Y 497.084,Z 462.247,A -85,B 0,C 180,E1 -6173.572,E2 -6173.572} C_VEL
LIN {X 0,Y 497.258,Z 466.061,A -85,B 0,C 180,E1 -6175.059,E2 -6175.059} C_VEL
LIN {X 0,Y 496.802,Z 475.164,A -85,B 0,C 180,E1 -6178.438,E2 -6178.438} C_VEL
LIN {X 0,Y 496.421,Z 484.458,A -85,B 0,C 180,E1 -6181.761,E2 -6181.761} C_VEL
LIN {X 0,Y 496.063,Z 494.019,A -85,B 0,C 180,E1 -6185.057,E2 -6185.057} C_VEL
LIN {X 0,Y 495.769,Z 503.928,A -85,B 0,C 180,E1 -6188.372,E2 -6188.372} C_VEL
LIN {X 0,Y 495.574,Z 513.186,A -85,B 0,C 180,E1 -6191.392,E2 -6191.392} C_VEL
LIN {X 0,Y 495.403,Z 523.638,A -85,B 0,C 180,E1 -6194.727,E2 -6194.727} C_VEL
LIN {X 0,Y 495.352,Z 526.042,A -85,B 0,C 180,E1 -6195.493,E2 -6195.493} C_VEL
LIN {X 0,Y 497.532,Z 540.946,A -85,B 0,C 180,E1 -6195.949,E2 -6195.949} C_VEL
LIN {X 0,Y 497.352,Z 553.965,A -85,B 0,C 180,E1 -6196.465,E2 -6196.465} C_VEL
LIN {X 0,Y 496.994,Z 566.049,A -85,B 0,C 180,E1 -6197.11,E2 -6197.11} C_VEL
LIN {X 0,Y 496.614,Z 576.826,A -85,B 0,C 180,E1 -6197.848,E2 -6197.848} C_VEL
LIN {X 0,Y 496.248,Z 587.614,A -85,B 0,C 180,E1 -6198.771,E2 -6198.771} C_VEL
LIN {X 0,Y 495.847,Z 597.332,A -85,B 0,C 180,E1 -6199.795,E2 -6199.795} C_VEL
LIN {X 0,Y 495.587,Z 605.319,A -85,B 0,C 180,E1 -6200.82,E2 -6200.82} C_VEL
LIN {X 0,Y 495.358,Z 613.135,A -85,B 0,C 180,E1 -6202.049,E2 -6202.049} C_VEL
LIN {X 0,Y 495.253,Z 618.475,A -85,B 0,C 180,E1 -6203.072,E2 -6203.072} C_VEL
LIN {X 0,Y 495.154,Z 623.657,A -85,B 0,C 180,E1 -6204.298,E2 -6204.298} C_VEL
LIN {X 0,Y 495.027,Z 627.67,A -85,B 0,C 180,E1 -6205.521,E2 -6205.521} C_VEL
LIN {X 0,Y 495.044,Z 630.635,A -85,B 0,C 180,E1 -6206.745,E2 -6206.745} C_VEL
LIN {X 0,Y 495.053,Z 632.049,A -85,B 0,C 180,E1 -6207.559,E2 -6207.559} C_VEL
LIN {X 0,Y 494.91,Z 633.653,A -85,B 0,C 180,E1 -6209.186,E2 -6209.186} C_VEL
LIN {X 0,Y 494.898,Z 633.862,A -85,B 0,C 180,E1 -6210,E2 -6210} C_VEL
LIN {X 0,Y 494.963,Z 633.014,A -85,B 0,C 180,E1 -6211.627,E2 -6211.627} C_VEL
LIN {X 0,Y 495.053,Z 631.995,A -85,B 0,C 180,E1 -6212.441,E2 -6212.441} C_VEL
LIN {X 0,Y 495.044,Z 630.558,A -85,B 0,C 180,E1 -6213.255,E2 -6213.255} C_VEL
LIN {X 0,Y 495.028,Z 627.551,A -85,B 0,C 180,E1 -6214.478,E2 -6214.478} C_VEL
LIN {X 0,Y 495.154,Z 623.491,A -85,B 0,C 180,E1 -6215.702,E2 -6215.702} C_VEL
LIN {X 0,Y 495.257,Z 617.239,A -85,B 0,C 180,E1 -6217.133,E2 -6217.133} C_VEL
LIN {X 0,Y 495.443,Z 610.411,A -85,B 0,C 180,E1 -6218.36,E2 -6218.36} C_VEL
LIN {X 0,Y 495.654,Z 601.927,A -85,B 0,C 180,E1 -6219.591,E2 -6219.591} C_VEL
LIN {X 0,Y 495.996,Z 593.216,A -85,B 0,C 180,E1 -6220.615,E2 -6220.615} C_VEL
LIN {X 0,Y 496.301,Z 582.485,A -85,B 0,C 180,E1 -6221.642,E2 -6221.642} C_VEL
LIN {X 0,Y 496.724,Z 571.216,A -85,B 0,C 180,E1 -6222.509,E2 -6222.509} C_VEL
LIN {X 0,Y 497.059,Z 560.223,A -85,B 0,C 180,E1 -6223.179,E2 -6223.179} C_VEL
LIN {X 0,Y 497.404,Z 546.966,A -85,B 0,C 180,E1 -6223.794,E2 -6223.794} C_VEL
LIN {X 0,Y 497.37,Z 540.235,A -85,B 0,C 180,E1 -6224.043,E2 -6224.043} C_VEL
LIN {X 0,Y 495.602,Z 527.763,A -85,B 0,C 180,E1 -6224.428,E2 -6224.428} C_VEL
LIN {X 0,Y 495.333,Z 525.174,A -85,B 0,C 180,E1 -6224.508,E2 -6224.508} C_VEL
LIN {X 0,Y 495.409,Z 515.995,A -85,B 0,C 180,E1 -6227.332,E2 -6227.332} C_VEL
LIN {X 0,Y 495.608,Z 505.5,A -85,B 0,C 180,E1 -6230.623,E2 -6230.623} C_VEL
LIN {X 0,Y 495.8,Z 495.614,A -85,B 0,C 180,E1 -6233.828,E2 -6233.828} C_VEL
LIN {X 0,Y 496.08,Z 486.42,A -85,B 0,C 180,E1 -6236.959,E2 -6236.959} C_VEL
LIN {X 0,Y 496.452,Z 477.352,A -85,B 0,C 180,E1 -6240.283,E2 -6240.283} C_VEL
LIN {X 0,Y 496.938,Z 469.518,A -85,B 0,C 180,E1 -6243.474,E2 -6243.474} C_VEL
LIN {X 0,Y 497.272,Z 465.304,A -85,B 0,C 180,E1 -6245.413,E2 -6245.413} C_VEL
LIN {X 0,Y 496.987,Z 461.53,A -85,B 0,C 180,E1 -6247.45,E2 -6247.45} C_VEL
LIN {X 0,Y 496.29,Z 457.693,A -85,B 0,C 180,E1 -6250.12,E2 -6250.12} C_VEL
LIN {X 0,Y 495.838,Z 455.296,A -85,B 0,C 180,E1 -6252.519,E2 -6252.519} C_VEL
LIN {X 0,Y 495.737,Z 454.737,A -85,B 0,C 180,E1 -6254.001,E2 -6254.001} C_VEL
LIN {X 0,Y 495.736,Z 454.737,A -85,B 0,C 180,E1 -6257.118,E2 -6257.118} C_VEL
LIN {X 0,Y 495.762,Z 454.734,A -85,B 0,C 180,E1 -6259.953,E2 -6259.953} C_VEL
LIN {X 0,Y 495.735,Z 454.847,A -85,B 0,C 180,E1 -6262.553,E2 -6262.553} C_VEL
LIN {X 0,Y 495.852,Z 456.446,A -85,B 0,C 180,E1 -6265.293,E2 -6265.293} C_VEL
LIN {X 0,Y 495.707,Z 458.673,A -85,B 0,C 180,E1 -6268.36,E2 -6268.36} C_VEL
LIN {X 0,Y 495.568,Z 461.244,A -85,B 0,C 180,E1 -6271.554,E2 -6271.554} C_VEL
LIN {X 0,Y 495.445,Z 463.296,A -85,B 0,C 180,E1 -6273.913,E2 -6273.913} C_VEL
LIN {X 0,Y 495.354,Z 465.717,A -85,B 0,C 180,E1 -6276.593,E2 -6276.593} C_VEL
LIN {X 0,Y 495.295,Z 468.43,A -85,B 0,C 180,E1 -6279.474,E2 -6279.474} C_VEL
LIN {X 0,Y 495.197,Z 471.563,A -85,B 0,C 180,E1 -6282.66,E2 -6282.66} C_VEL
LIN {X 0,Y 495.182,Z 474.603,A -85,B 0,C 180,E1 -6285.645,E2 -6285.645} C_VEL
LIN {X 0,Y 497.513,Z 486.029,A -85,B 0,C 180,E1 -6286.053,E2 -6286.053} C_VEL
LIN {X 0,Y 497.498,Z 497.507,A -85,B 0,C 180,E1 -6286.521,E2 -6286.521} C_VEL
LIN {X 0,Y 497.18,Z 509.421,A -85,B 0,C 180,E1 -6287.158,E2 -6287.158} C_VEL
LIN {X 0,Y 496.827,Z 520.969,A -85,B 0,C 180,E1 -6287.957,E2 -6287.957} C_VEL
LIN {X 0,Y 496.403,Z 531.549,A -85,B 0,C 180,E1 -6288.878,E2 -6288.878} C_VEL
LIN {X 0,Y 496.1,Z 540.2,A -85,B 0,C 180,E1 -6289.8,E2 -6289.8} C_VEL
LIN {X 0,Y 495.837,Z 548.154,A -85,B 0,C 180,E1 -6290.825,E2 -6290.825} C_VEL
LIN {X 0,Y 495.519,Z 555.948,A -85,B 0,C 180,E1 -6292.052,E2 -6292.052} C_VEL
LIN {X 0,Y 495.305,Z 562.419,A -85,B 0,C 180,E1 -6293.34,E2 -6293.34} C_VEL
LIN {X 0,Y 495.129,Z 567.772,A -85,B 0,C 180,E1 -6294.706,E2 -6294.706} C_VEL
LIN {X 0,Y 495.17,Z 571.38,A -85,B 0,C 180,E1 -6295.931,E2 -6295.931} C_VEL
LIN {X 0,Y 495.062,Z 573.246,A -85,B 0,C 180,E1 -6296.745,E2 -6296.745} C_VEL
LIN {X 0,Y 495.055,Z 574.654,A -85,B 0,C 180,E1 -6297.559,E2 -6297.559} C_VEL
LIN {X 0,Y 494.911,Z 576.258,A -85,B 0,C 180,E1 -6299.187,E2 -6299.187} C_VEL
LIN {X 0,Y 494.899,Z 576.482,A -85,B 0,C 180,E1 -6300,E2 -6300} C_VEL
LIN {X 0,Y 494.911,Z 576.285,A -85,B 0,C 180,E1 -6300.814,E2 -6300.814} C_VEL
LIN {X 0,Y 495.054,Z 574.695,A -85,B 0,C 180,E1 -6302.441,E2 -6302.441} C_VEL
LIN {X 0,Y 495.051,Z 573.319,A -85,B 0,C 180,E1 -6303.256,E2 -6303.256} C_VEL
LIN {X 0,Y 495.138,Z 570.417,A -85,B 0,C 180,E1 -6304.478,E2 -6304.478} C_VEL
LIN {X 0,Y 495.229,Z 566.487,A -85,B 0,C 180,E1 -6305.701,E2 -6305.701} C_VEL
LIN {X 0,Y 495.357,Z 561.421,A -85,B 0,C 180,E1 -6306.926,E2 -6306.926} C_VEL
LIN {X 0,Y 495.515,Z 555.029,A -85,B 0,C 180,E1 -6308.154,E2 -6308.154} C_VEL
LIN {X 0,Y 495.762,Z 547.044,A -85,B 0,C 180,E1 -6309.383,E2 -6309.383} C_VEL
LIN {X 0,Y 496.113,Z 538.896,A -85,B 0,C 180,E1 -6310.406,E2 -6310.406} C_VEL
LIN {X 0,Y 496.508,Z 528.962,A -85,B 0,C 180,E1 -6311.43,E2 -6311.43} C_VEL
LIN {X 0,Y 496.87,Z 518.15,A -85,B 0,C 180,E1 -6312.323,E2 -6312.323} C_VEL
LIN {X 0,Y 497.173,Z 506.78,A -85,B 0,C 180,E1 -6313.072,E2 -6313.072} C_VEL
LIN {X 0,Y 497.538,Z 494.706,A -85,B 0,C 180,E1 -6313.686,E2 -6313.686} C_VEL
LIN {X 0,Y 497.542,Z 486.464,A -85,B 0,C 180,E1 -6314.012,E2 -6314.012} C_VEL
LIN {X 0,Y 495.668,Z 476.279,A -85,B 0,C 180,E1 -6314.376,E2 -6314.376} C_VEL
LIN {X 0,Y 495.086,Z 473.507,A -85,B 0,C 180,E1 -6314.473,E2 -6314.473} C_VEL
LIN {X 0,Y 495.1,Z 469.55,A -85,B 0,C 180,E1 -6317.996,E2 -6317.996} C_VEL
LIN {X 0,Y 495.096,Z 466.462,A -85,B 0,C 180,E1 -6320.786,E2 -6320.786} C_VEL
LIN {X 0,Y 495.14,Z 463.562,A -85,B 0,C 180,E1 -6323.418,E2 -6323.418} C_VEL
LIN {X 0,Y 495.238,Z 460.102,A -85,B 0,C 180,E1 -6326.614,E2 -6326.614} C_VEL
LIN {X 0,Y 495.278,Z 456.402,A -85,B 0,C 180,E1 -6330.049,E2 -6330.049} C_VEL
LIN {X 0,Y 495.269,Z 454.797,A -85,B 0,C 180,E1 -6331.671,E2 -6331.671} C_VEL
LIN {X 0,Y 495.654,Z 454.748,A -85,B 0,C 180,E1 -6334.674,E2 -6334.674} C_VEL
LIN {X 0,Y 495.724,Z 454.735,A -85,B 0,C 180,E1 -6337.563,E2 -6337.563} C_VEL
LIN {X 0,Y 495.763,Z 454.731,A -85,B 0,C 180,E1 -6340.047,E2 -6340.047} C_VEL
LIN {X 0,Y 495.738,Z 454.732,A -85,B 0,C 180,E1 -6342.882,E2 -6342.882} C_VEL
LIN {X 0,Y 495.739,Z 454.734,A -85,B 0,C 180,E1 -6345.999,E2 -6345.999} C_VEL
LIN {X 0,Y 495.771,Z 454.731,A -85,B 0,C 180,E1 -6349.3,E2 -6349.3} C_VEL
LIN {X 0,Y 495.734,Z 454.737,A -85,B 0,C 180,E1 -6352.439,E2 -6352.439} C_VEL
LIN {X 0,Y 495.784,Z 454.727,A -85,B 0,C 180,E1 -6355.457,E2 -6355.457} C_VEL
LIN {X 0,Y 495.797,Z 454.725,A -85,B 0,C 180,E1 -6356.768,E2 -6356.768} C_VEL
LIN {X 0,Y 495.093,Z 454.816,A -85,B 0,C 180,E1 -6357.445,E2 -6357.445} C_VEL
LIN {X 0,Y 492.216,Z 455.172,A -85,B 0,C 180,E1 -6358.545,E2 -6358.545} C_VEL
LIN {X 0,Y 489.811,Z 455.474,A -85,B 0,C 180,E1 -6359.432,E2 -6359.432} C_VEL
LIN {X 0,Y 488.791,Z 455.598,A -85,B 0,C 180,E1 -6360.117,E2 -6360.117} C_VEL
LIN {X 0,Y 488.713,Z 455.608,A -85,B 0,C 180,E1 -6360.348,E2 -6360.348} C_VEL
LIN {X 0,Y 488.797,Z 455.599,A -85,B 0,C 180,E1 -6363.057,E2 -6363.057} C_VEL
LIN {X 0,Y 488.686,Z 455.615,A -85,B 0,C 180,E1 -6366.254,E2 -6366.254} C_VEL
LIN {X 0,Y 488.752,Z 455.604,A -85,B 0,C 180,E1 -6369.176,E2 -6369.176} C_VEL
LIN {X 0,Y 488.755,Z 455.605,A -85,B 0,C 180,E1 -6371.632,E2 -6371.632} C_VEL
LIN {X 0,Y 488.768,Z 455.603,A -85,B 0,C 180,E1 -6375,E2 -6375} C_VEL
LIN {X 0,Y 488.812,Z 455.597,A -85,B 0,C 180,E1 -6378.388,E2 -6378.388} C_VEL
LIN {X 0,Y 488.822,Z 455.599,A -85,B 0,C 180,E1 -6381.734,E2 -6381.734} C_VEL
LIN {X 0,Y 488.859,Z 455.59,A -85,B 0,C 180,E1 -6384.224,E2 -6384.224} C_VEL
LIN {X 0,Y 488.967,Z 455.576,A -85,B 0,C 180,E1 -6387.529,E2 -6387.529} C_VEL
LIN {X 0,Y 488.94,Z 455.578,A -85,B 0,C 180,E1 -6390.824,E2 -6390.824} C_VEL
LIN {X 0,Y 488.967,Z 455.576,A -85,B 0,C 180,E1 -6392.471,E2 -6392.471} C_VEL
LIN {X 0,Y 488.845,Z 455.593,A -85,B 0,C 180,E1 -6395.776,E2 -6395.776} C_VEL
LIN {X 0,Y 488.791,Z 455.599,A -85,B 0,C 180,E1 -6398.267,E2 -6398.267} C_VEL
LIN {X 0,Y 488.812,Z 455.595,A -85,B 0,C 180,E1 -6401.612,E2 -6401.612} C_VEL
LIN {X 0,Y 488.768,Z 455.6,A -85,B 0,C 180,E1 -6405,E2 -6405} C_VEL
LIN {X 0,Y 488.761,Z 455.602,A -85,B 0,C 180,E1 -6408.442,E2 -6408.442} C_VEL
LIN {X 0,Y 488.712,Z 455.611,A -85,B 0,C 180,E1 -6411.071,E2 -6411.071} C_VEL
LIN {X 0,Y 488.686,Z 455.612,A -85,B 0,C 180,E1 -6413.746,E2 -6413.746} C_VEL
LIN {X 0,Y 488.797,Z 455.595,A -85,B 0,C 180,E1 -6416.943,E2 -6416.943} C_VEL
LIN {X 0,Y 488.715,Z 455.607,A -85,B 0,C 180,E1 -6420.363,E2 -6420.363} C_VEL
LIN {X 0,Y 488.741,Z 455.605,A -85,B 0,C 180,E1 -6423.484,E2 -6423.484} C_VEL
LIN {X 0,Y 488.693,Z 455.612,A -85,B 0,C 180,E1 -6426.355,E2 -6426.355} C_VEL
LIN {X 0,Y 488.705,Z 455.608,A -85,B 0,C 180,E1 -6429.254,E2 -6429.254} C_VEL
LIN {X 0,Y 488.712,Z 455.611,A -85,B 0,C 180,E1 -6431.6,E2 -6431.6} C_VEL
LIN {X 0,Y 488.717,Z 455.61,A -85,B 0,C 180,E1 -6434.801,E2 -6434.801} C_VEL
LIN {X 0,Y 488.7,Z 455.609,A -85,B 0,C 180,E1 -6437.475,E2 -6437.475} C_VEL
LIN {X 0,Y 488.737,Z 455.607,A -85,B 0,C 180,E1 -6439.676,E2 -6439.676} C_VEL
LIN {X 0,Y 488.681,Z 455.611,A -85,B 0,C 180,E1 -6442.841,E2 -6442.841} C_VEL
LIN {X 0,Y 488.564,Z 455.631,A -85,B 0,C 180,E1 -6445.873,E2 -6445.873} C_VEL
LIN {X 0,Y 488.231,Z 455.672,A -85,B 0,C 180,E1 -6448.787,E2 -6448.787} C_VEL
LIN {X 0,Y 488.096,Z 455.689,A -85,B 0,C 180,E1 -6449.761,E2 -6449.761} C_VEL
LIN {X 0,Y 488.121,Z 459.663,A -85,B 0,C 180,E1 -6453.213,E2 -6453.213} C_VEL
LIN {X 0,Y 488.037,Z 463.123,A -85,B 0,C 180,E1 -6456.22,E2 -6456.22} C_VEL
LIN {X 0,Y 488.028,Z 467.233,A -85,B 0,C 180,E1 -6459.78,E2 -6459.78} C_VEL
LIN {X 0,Y 487.986,Z 470.221,A -85,B 0,C 180,E1 -6462.395,E2 -6462.395} C_VEL
LIN {X 0,Y 488.012,Z 473.847,A -85,B 0,C 180,E1 -6465.433,E2 -6465.433} C_VEL
LIN {X 0,Y 490.344,Z 485.213,A -85,B 0,C 180,E1 -6465.83,E2 -6465.83} C_VEL
LIN {X 0,Y 490.747,Z 489.873,A -85,B 0,C 180,E1 -6466.015,E2 -6466.015} C_VEL
LIN {X 0,Y 490.422,Z 501.406,A -85,B 0,C 180,E1 -6466.534,E2 -6466.534} C_VEL
LIN {X 0,Y 490.095,Z 513.366,A -85,B 0,C 180,E1 -6467.247,E2 -6467.247} C_VEL
LIN {X 0,Y 489.739,Z 524.515,A -85,B 0,C 180,E1 -6468.095,E2 -6468.095} C_VEL
LIN {X 0,Y 489.299,Z 534.463,A -85,B 0,C 180,E1 -6469.029,E2 -6469.029} C_VEL
LIN {X 0,Y 488.942,Z 543.448,A -85,B 0,C 180,E1 -6470.067,E2 -6470.067} C_VEL
LIN {X 0,Y 488.614,Z 552.2,A -85,B 0,C 180,E1 -6471.313,E2 -6471.313} C_VEL
LIN {X 0,Y 488.348,Z 559.245,A -85,B 0,C 180,E1 -6472.558,E2 -6472.558} C_VEL
LIN {X 0,Y 488.223,Z 565.314,A -85,B 0,C 180,E1 -6473.924,E2 -6473.924} C_VEL
LIN {X 0,Y 488.074,Z 570.468,A -85,B 0,C 180,E1 -6475.457,E2 -6475.457} C_VEL
LIN {X 0,Y 487.98,Z 573.452,A -85,B 0,C 180,E1 -6476.697,E2 -6476.697} C_VEL
LIN {X 0,Y 487.989,Z 574.905,A -85,B 0,C 180,E1 -6477.523,E2 -6477.523} C_VEL
LIN {X 0,Y 487.834,Z 576.573,A -85,B 0,C 180,E1 -6479.174,E2 -6479.174} C_VEL
LIN {X 0,Y 487.821,Z 576.83,A -85,B 0,C 180,E1 -6480,E2 -6480} C_VEL
LIN {X 0,Y 487.834,Z 576.655,A -85,B 0,C 180,E1 -6480.825,E2 -6480.825} C_VEL
LIN {X 0,Y 487.99,Z 575.121,A -85,B 0,C 180,E1 -6482.476,E2 -6482.476} C_VEL
LIN {X 0,Y 487.99,Z 573.763,A -85,B 0,C 180,E1 -6483.302,E2 -6483.302} C_VEL
LIN {X 0,Y 488.072,Z 570.896,A -85,B 0,C 180,E1 -6484.542,E2 -6484.542} C_VEL
LIN {X 0,Y 488.222,Z 565.858,A -85,B 0,C 180,E1 -6486.082,E2 -6486.082} C_VEL
LIN {X 0,Y 488.353,Z 559.951,A -85,B 0,C 180,E1 -6487.442,E2 -6487.442} C_VEL
LIN {X 0,Y 488.629,Z 553.062,A -85,B 0,C 180,E1 -6488.686,E2 -6488.686} C_VEL
LIN {X 0,Y 488.923,Z 544.465,A -85,B 0,C 180,E1 -6489.933,E2 -6489.933} C_VEL
LIN {X 0,Y 489.296,Z 535.648,A -85,B 0,C 180,E1 -6490.971,E2 -6490.971} C_VEL
LIN {X 0,Y 489.704,Z 525.902,A -85,B 0,C 180,E1 -6491.906,E2 -6491.906} C_VEL
LIN {X 0,Y 490.037,Z 513.859,A -85,B 0,C 180,E1 -6492.832,E2 -6492.832} C_VEL
LIN {X 0,Y 490.451,Z 501.36,A -85,B 0,C 180,E1 -6493.571,E2 -6493.571} C_VEL
LIN {X 0,Y 490.777,Z 488.354,A -85,B 0,C 180,E1 -6494.143,E2 -6494.143} C_VEL
LIN {X 0,Y 489.229,Z 479.714,A -85,B 0,C 180,E1 -6494.474,E2 -6494.474} C_VEL
LIN {X 0,Y 488.096,Z 474.754,A -85,B 0,C 180,E1 -6494.648,E2 -6494.648} C_VEL
LIN {X 0,Y 488.098,Z 470.742,A -85,B 0,C 180,E1 -6498.136,E2 -6498.136} C_VEL
LIN {X 0,Y 488.077,Z 467.275,A -85,B 0,C 180,E1 -6501.099,E2 -6501.099} C_VEL
LIN {X 0,Y 488.099,Z 464.137,A -85,B 0,C 180,E1 -6503.776,E2 -6503.776} C_VEL
LIN {X 0,Y 488.153,Z 460.246,A -85,B 0,C 180,E1 -6506.795,E2 -6506.795} C_VEL
LIN {X 0,Y 488.117,Z 455.688,A -85,B 0,C 180,E1 -6510.261,E2 -6510.261} C_VEL
LIN {X 0,Y 488.488,Z 455.641,A -85,B 0,C 180,E1 -6513.142,E2 -6513.142} C_VEL
LIN {X 0,Y 488.642,Z 455.619,A -85,B 0,C 180,E1 -6515.121,E2 -6515.121} C_VEL
LIN {X 0,Y 488.682,Z 455.616,A -85,B 0,C 180,E1 -6518.2,E2 -6518.2} C_VEL
LIN {X 0,Y 488.721,Z 455.609,A -85,B 0,C 180,E1 -6521.414,E2 -6521.414} C_VEL
LIN {X 0,Y 488.705,Z 455.611,A -85,B 0,C 180,E1 -6524.024,E2 -6524.024} C_VEL
LIN {X 0,Y 488.712,Z 455.612,A -85,B 0,C 180,E1 -6527.173,E2 -6527.173} C_VEL
LIN {X 0,Y 488.735,Z 455.655,A -85,B 0,C 180,E1 -6530.215,E2 -6530.215} C_VEL
LIN {X 0,Y 490.076,Z 463.272,A -85,B 0,C 180,E1 -6533.425,E2 -6533.425} C_VEL
LIN {X 0,Y 490.272,Z 467.269,A -85,B 0,C 180,E1 -6535.012,E2 -6535.012} C_VEL
LIN {X 0,Y 489.862,Z 475.022,A -85,B 0,C 180,E1 -6537.938,E2 -6537.938} C_VEL
LIN {X 0,Y 489.434,Z 483.842,A -85,B 0,C 180,E1 -6541.155,E2 -6541.155} C_VEL
LIN {X 0,Y 489.128,Z 491.912,A -85,B 0,C 180,E1 -6544.008,E2 -6544.008} C_VEL
LIN {X 0,Y 488.8,Z 501.073,A -85,B 0,C 180,E1 -6547.157,E2 -6547.157} C_VEL
LIN {X 0,Y 488.56,Z 510.29,A -85,B 0,C 180,E1 -6550.242,E2 -6550.242} C_VEL
LIN {X 0,Y 488.407,Z 518.204,A -85,B 0,C 180,E1 -6552.843,E2 -6552.843} C_VEL
LIN {X 0,Y 488.288,Z 525.721,A -85,B 0,C 180,E1 -6555.278,E2 -6555.278} C_VEL
LIN {X 0,Y 490.535,Z 541.154,A -85,B 0,C 180,E1 -6555.771,E2 -6555.771} C_VEL
LIN {X 0,Y 490.416,Z 553.413,A -85,B 0,C 180,E1 -6556.27,E2 -6556.27} C_VEL
LIN {X 0,Y 490.034,Z 564.296,A -85,B 0,C 180,E1 -6556.85,E2 -6556.85} C_VEL
LIN {X 0,Y 489.63,Z 576.321,A -85,B 0,C 180,E1 -6557.672,E2 -6557.672} C_VEL
LIN {X 0,Y 489.254,Z 587.124,A -85,B 0,C 180,E1 -6558.608,E2 -6558.608} C_VEL
LIN {X 0,Y 488.822,Z 596.857,A -85,B 0,C 180,E1 -6559.647,E2 -6559.647} C_VEL
LIN {X 0,Y 488.518,Z 604.857,A -85,B 0,C 180,E1 -6560.686,E2 -6560.686} C_VEL
LIN {X 0,Y 488.292,Z 612.695,A -85,B 0,C 180,E1 -6561.933,E2 -6561.933} C_VEL
LIN {X 0,Y 488.069,Z 619.885,A -85,B 0,C 180,E1 -6563.385,E2 -6563.385} C_VEL
LIN {X 0,Y 488.052,Z 624.682,A -85,B 0,C 180,E1 -6564.629,E2 -6564.629} C_VEL
LIN {X 0,Y 487.958,Z 628.34,A -85,B 0,C 180,E1 -6565.87,E2 -6565.87} C_VEL
LIN {X 0,Y 487.968,Z 630.228,A -85,B 0,C 180,E1 -6566.697,E2 -6566.697} C_VEL
LIN {X 0,Y 487.959,Z 631.643,A -85,B 0,C 180,E1 -6567.524,E2 -6567.524} C_VEL
LIN {X 0,Y 487.893,Z 632.644,A -85,B 0,C 180,E1 -6568.349,E2 -6568.349} C_VEL
LIN {X 0,Y 487.819,Z 633.453,A -85,B 0,C 180,E1 -6570,E2 -6570} C_VEL
LIN {X 0,Y 487.893,Z 632.597,A -85,B 0,C 180,E1 -6571.651,E2 -6571.651} C_VEL
LIN {X 0,Y 487.972,Z 631.567,A -85,B 0,C 180,E1 -6572.476,E2 -6572.476} C_VEL
LIN {X 0,Y 487.969,Z 630.122,A -85,B 0,C 180,E1 -6573.303,E2 -6573.303} C_VEL
LIN {X 0,Y 487.937,Z 627.097,A -85,B 0,C 180,E1 -6574.544,E2 -6574.544} C_VEL
LIN {X 0,Y 488.05,Z 623.014,A -85,B 0,C 180,E1 -6575.785,E2 -6575.785} C_VEL
LIN {X 0,Y 488.182,Z 616.735,A -85,B 0,C 180,E1 -6577.237,E2 -6577.237} C_VEL
LIN {X 0,Y 488.368,Z 609.87,A -85,B 0,C 180,E1 -6578.482,E2 -6578.482} C_VEL
LIN {X 0,Y 488.601,Z 601.352,A -85,B 0,C 180,E1 -6579.73,E2 -6579.73} C_VEL
LIN {X 0,Y 488.949,Z 592.6,A -85,B 0,C 180,E1 -6580.77,E2 -6580.77} C_VEL
LIN {X 0,Y 489.307,Z 581.832,A -85,B 0,C 180,E1 -6581.811,E2 -6581.811} C_VEL
LIN {X 0,Y 489.732,Z 570.333,A -85,B 0,C 180,E1 -6582.703,E2 -6582.703} C_VEL
LIN {X 0,Y 490.116,Z 559.472,A -85,B 0,C 180,E1 -6583.369,E2 -6583.369} C_VEL
LIN {X 0,Y 490.512,Z 546.206,A -85,B 0,C 180,E1 -6583.992,E2 -6583.992} C_VEL
LIN {X 0,Y 490.368,Z 540.922,A -85,B 0,C 180,E1 -6584.195,E2 -6584.195} C_VEL
LIN {X 0,Y 488.518,Z 527.255,A -85,B 0,C 180,E1 -6584.635,E2 -6584.635} C_VEL
LIN {X 0,Y 488.24,Z 524.74,A -85,B 0,C 180,E1 -6584.697,E2 -6584.697} C_VEL
LIN {X 0,Y 488.317,Z 515.514,A -85,B 0,C 180,E1 -6587.592,E2 -6587.592} C_VEL
LIN {X 0,Y 488.542,Z 505.628,A -85,B 0,C 180,E1 -6590.76,E2 -6590.76} C_VEL
LIN {X 0,Y 488.738,Z 496.62,A -85,B 0,C 180,E1 -6593.743,E2 -6593.743} C_VEL
LIN {X 0,Y 489.05,Z 487.257,A -85,B 0,C 180,E1 -6597.003,E2 -6597.003} C_VEL
LIN {X 0,Y 489.394,Z 478.773,A -85,B 0,C 180,E1 -6600.174,E2 -6600.174} C_VEL
LIN {X 0,Y 489.855,Z 471.837,A -85,B 0,C 180,E1 -6603.038,E2 -6603.038} C_VEL
LIN {X 0,Y 490.28,Z 467.136,A -85,B 0,C 180,E1 -6605.207,E2 -6605.207} C_VEL
LIN {X 0,Y 490.124,Z 463.758,A -85,B 0,C 180,E1 -6607.031,E2 -6607.031} C_VEL
LIN {X 0,Y 489.602,Z 460.473,A -85,B 0,C 180,E1 -6609.182,E2 -6609.182} C_VEL
LIN {X 0,Y 489.068,Z 457.644,A -85,B 0,C 180,E1 -6611.647,E2 -6611.647} C_VEL
LIN {X 0,Y 488.735,Z 455.882,A -85,B 0,C 180,E1 -6614.028,E2 -6614.028} C_VEL
LIN {X 0,Y 488.695,Z 455.614,A -85,B 0,C 180,E1 -6616.346,E2 -6616.346} C_VEL
LIN {X 0,Y 488.722,Z 455.611,A -85,B 0,C 180,E1 -6618.586,E2 -6618.586} C_VEL
LIN {X 0,Y 488.711,Z 455.794,A -85,B 0,C 180,E1 -6621.803,E2 -6621.803} C_VEL
LIN {X 0,Y 488.84,Z 456.779,A -85,B 0,C 180,E1 -6623.882,E2 -6623.882} C_VEL
LIN {X 0,Y 488.765,Z 458.661,A -85,B 0,C 180,E1 -6626.879,E2 -6626.879} C_VEL
LIN {X 0,Y 488.624,Z 460.804,A -85,B 0,C 180,E1 -6629.774,E2 -6629.774} C_VEL
LIN {X 0,Y 488.475,Z 463.083,A -85,B 0,C 180,E1 -6632.587,E2 -6632.587} C_VEL
LIN {X 0,Y 488.382,Z 465.456,A -85,B 0,C 180,E1 -6635.334,E2 -6635.334} C_VEL
LIN {X 0,Y 488.245,Z 467.905,A -85,B 0,C 180,E1 -6638.022,E2 -6638.022} C_VEL
LIN {X 0,Y 488.153,Z 470.399,A -85,B 0,C 180,E1 -6640.662,E2 -6640.662} C_VEL
LIN {X 0,Y 488.139,Z 472.939,A -85,B 0,C 180,E1 -6643.265,E2 -6643.265} C_VEL
LIN {X 0,Y 488.17,Z 475.331,A -85,B 0,C 180,E1 -6645.449,E2 -6645.449} C_VEL
LIN {X 0,Y 490.613,Z 486.669,A -85,B 0,C 180,E1 -6645.866,E2 -6645.866} C_VEL
LIN {X 0,Y 490.631,Z 496.663,A -85,B 0,C 180,E1 -6646.276,E2 -6646.276} C_VEL
LIN {X 0,Y 490.277,Z 508.534,A -85,B 0,C 180,E1 -6646.905,E2 -6646.905} C_VEL
LIN {X 0,Y 489.935,Z 519.912,A -85,B 0,C 180,E1 -6647.68,E2 -6647.68} C_VEL
LIN {X 0,Y 489.486,Z 530.798,A -85,B 0,C 180,E1 -6648.614,E2 -6648.614} C_VEL
LIN {X 0,Y 489.119,Z 540.531,A -85,B 0,C 180,E1 -6649.653,E2 -6649.653} C_VEL
LIN {X 0,Y 488.836,Z 548.506,A -85,B 0,C 180,E1 -6650.692,E2 -6650.692} C_VEL
LIN {X 0,Y 488.504,Z 556.323,A -85,B 0,C 180,E1 -6651.937,E2 -6651.937} C_VEL
LIN {X 0,Y 488.265,Z 563.073,A -85,B 0,C 180,E1 -6653.304,E2 -6653.304} C_VEL
LIN {X 0,Y 488.074,Z 568.177,A -85,B 0,C 180,E1 -6654.63,E2 -6654.63} C_VEL
LIN {X 0,Y 488.106,Z 571.792,A -85,B 0,C 180,E1 -6655.872,E2 -6655.872} C_VEL
LIN {X 0,Y 487.99,Z 573.661,A -85,B 0,C 180,E1 -6656.698,E2 -6656.698} C_VEL
LIN {X 0,Y 487.99,Z 575.071,A -85,B 0,C 180,E1 -6657.524,E2 -6657.524} C_VEL
LIN {X 0,Y 487.834,Z 576.672,A -85,B 0,C 180,E1 -6659.175,E2 -6659.175} C_VEL
LIN {X 0,Y 487.82,Z 576.895,A -85,B 0,C 180,E1 -6660,E2 -6660} C_VEL
LIN {X 0,Y 487.834,Z 576.692,A -85,B 0,C 180,E1 -6660.826,E2 -6660.826} C_VEL
LIN {X 0,Y 487.989,Z 575.087,A -85,B 0,C 180,E1 -6662.477,E2 -6662.477} C_VEL
LIN {X 0,Y 487.98,Z 573.705,A -85,B 0,C 180,E1 -6663.303,E2 -6663.303} C_VEL
LIN {X 0,Y 488.069,Z 570.789,A -85,B 0,C 180,E1 -6664.543,E2 -6664.543} C_VEL
LIN {X 0,Y 488.178,Z 566.841,A -85,B 0,C 180,E1 -6665.784,E2 -6665.784} C_VEL
LIN {X 0,Y 488.336,Z 560.859,A -85,B 0,C 180,E1 -6667.214,E2 -6667.214} C_VEL
LIN {X 0,Y 488.55,Z 554.101,A -85,B 0,C 180,E1 -6668.479,E2 -6668.479} C_VEL
LIN {X 0,Y 488.841,Z 545.836,A -85,B 0,C 180,E1 -6669.726,E2 -6669.726} C_VEL
LIN {X 0,Y 489.152,Z 537.348,A -85,B 0,C 180,E1 -6670.765,E2 -6670.765} C_VEL
LIN {X 0,Y 489.664,Z 526.865,A -85,B 0,C 180,E1 -6671.802,E2 -6671.802} C_VEL
LIN {X 0,Y 489.97,Z 516.117,A -85,B 0,C 180,E1 -6672.665,E2 -6672.665} C_VEL
LIN {X 0,Y 490.306,Z 505.19,A -85,B 0,C 180,E1 -6673.364,E2 -6673.364} C_VEL
LIN {X 0,Y 490.7,Z 492.329,A -85,B 0,C 180,E1 -6673.987,E2 -6673.987} C_VEL
LIN {X 0,Y 490.558,Z 486.559,A -85,B 0,C 180,E1 -6674.216,E2 -6674.216} C_VEL
LIN {X 0,Y 488.41,Z 475.816,A -85,B 0,C 180,E1 -6674.607,E2 -6674.607} C_VEL
LIN {X 0,Y 488.018,Z 473.84,A -85,B 0,C 180,E1 -6674.677,E2 -6674.677} C_VEL
LIN {X 0,Y 488.035,Z 469.992,A -85,B 0,C 180,E1 -6678.113,E2 -6678.113} C_VEL
LIN {X 0,Y 488.014,Z 466.694,A -85,B 0,C 180,E1 -6681.102,E2 -6681.102} C_VEL
LIN {X 0,Y 488.065,Z 463.778,A -85,B 0,C 180,E1 -6683.778,E2 -6683.778} C_VEL
LIN {X 0,Y 488.172,Z 460.512,A -85,B 0,C 180,E1 -6686.799,E2 -6686.799} C_VEL
LIN {X 0,Y 488.218,Z 456.831,A -85,B 0,C 180,E1 -6690.254,E2 -6690.254} C_VEL
LIN {X 0,Y 488.179,Z 455.82,A -85,B 0,C 180,E1 -6691.217,E2 -6691.217} C_VEL
